// Поддержка соединения
TNC (IN:=NOT Asda.Connect, PT:=T#2S);

CASE CNT OF
0: // Начало работы
	STEP:=0;	// Сброс селектора
	Asda.IsInit:=FALSE;
	Asda.IsHoming:=FALSE;
	Asda.IsServo_ON:=FALSE;
	Asda.Pusk:=FALSE;
	Asda.P2_30:=0;
	Asda.P3_06:=0;
	Asda.E_CODE:=0;
	ALARM_TEST:=FALSE;
	DEL (IN:=FALSE);
	CNT:=10;
	
10: // Ожидание соединения
	Asda.text_id:=12;	// Ожидание соединения
	IF Asda.Connect THEN
		CNT:=20;
	END_IF

20: // Инициализация
	ASDA_INIT (CNT:=STEP);
	IF STEP=0 THEN
		CNT:=TERNAR_INT (Asda.IsInit, 30, 1000);
	END_IF

30: // Запись параметров
	ASDA_PARAMS (CNT:=STEP);
	IF STEP=0 THEN
		CNT:=100;
	END_IF

//////////////////////////////////////////////////////////////////////////////////////////////////
// О Ж И Д А Н И Е  К О М А Н Д Ы  И  Р А З О Г Р Е В А //////////////////////////////////////////
//////////////////////////////////////////////////////////////////////////////////////////////////
100: // Если ручная работа, переход на ручную, иначе Достигла ли температура ? 
	CNT:=PENTAR_INT (Asda.AllowManual, Asda.Block, 180, 110, 130);

110: // Если температура не достигнута, то проверим, включен ли сервопривод, если включен, то отключим
	CNT:=TERNAR_INT (NOT Asda.IsServo_ON, 100, 120);
	
120: // Отключим сервопривод при низких температурах
	ASDA_SERVO_OFF (CNT:=STEP);
	IF STEP=0 THEN
		CNT:=100;
	END_IF
	
130: // Если температура достигнута, то проверим, включен ли сервопривод, если выключен, то включим его
	CNT:=TERNAR_INT (NOT Asda.IsServo_ON, 140, 150);

140: // Включим сервопривод
	ASDA_SERVO_ON (CNT:=STEP);
	IF STEP=0 THEN
		CNT:=150;
	END_IF
	
150: // Проверим Homing, если нет, то выполним Homing
	CNT:=TERNAR_INT (NOT Asda.IsHoming, 160, 170);

160: // Если не было Homing то сделаем Homing
	ASDA_HOMING (CNT:=STEP);
	IF STEP=0 THEN
		CNT:=170;
	END_IF
	
170: // Проверка на запуск
	Asda.text_id:=0; // Индекс сообщения
	CNT:=TERNAR_INT (Asda.Pusk, 200, 100);
	
//////////////////////////////////////////////////////////////////////////////////////////////////
// Р У Ч Н О Й  Р Е Ж И М  ///////////////////////////////////////////////////////////////////////
//////////////////////////////////////////////////////////////////////////////////////////////////
180: // Ручная работа сервопривода - ожидание снятия флага ручной работы
	Asda.text_id:=14;						// Сообщение
	IF NOT Asda.AllowManual THEN
		CNT:=100;
	END_IF
	
//////////////////////////////////////////////////////////////////////////////////////////////////
// О С Н О В Н А Я  Р А Б О Т А //////////////////////////////////////////////////////////////////
//////////////////////////////////////////////////////////////////////////////////////////////////
200: // Пульсирование
	ASDA_PULSING (CNT:=STEP);
	IF STEP=0 THEN
		CNT:=TERNAR_INT (NOT Asda.Block, 210, 100);
	END_IF
	
210: // Парковка
	ASDA_PARKING (CNT:=STEP);
	IF STEP=0 THEN
		CNT:=100;	// На ожидание
	END_IF

//////////////////////////////////////////////////////////////////////////////////////////////////
// О Б Р А Б О Т К А  О Ш И Б О К ////////////////////////////////////////////////////////////////
//////////////////////////////////////////////////////////////////////////////////////////////////
1000: // Сброс
	Asda.DoPulsing:=FALSE;
	STEP:=0;
	DEL (IN:=FALSE);
	CNT:=1010;
	
1010: // Если нет аварии сервопривода, то останов
	CNT:=TERNAR_INT (NOT Asda.E_CODE.0, 1020, 1030);

1020: // Если нет аварии сервопривода, то экстренный стоп
	ASDA_STOP (CNT:=STEP);
	IF STEP=0 THEN
		CNT:=1030;
	END_IF
	
1030: // Ожидание сигнала ОБЩЕГО СБРОСА АВАРИИ или сброса аварии только сервопривода
	Asda.text_id:=10;		// Обработка ошибки
	IF SBROS_AVARII OR SBROS_AVARII_ASDA THEN
		CNT:=TERNAR_INT (Asda.E_CODE.0, 1040, 1050);
	END_IF
	
1040: // Сброс аварии сервопривода
	ASDA_SERVO_ON (CNT:=STEP);
	IF STEP=0 THEN
		CNT:=1050;
	END_IF

1050: // Небольшая задержка
	DEL (IN:=TRUE, PT:=T#1S);
	IF DEL.Q THEN
		DEL (IN:=FALSE);
		CNT:=1060;
	END_IF

1060: // Ожидание пропадания сигнала SBROS_AVARII
	IF NOT (SBROS_AVARII OR SBROS_AVARII_ASDA) THEN
		Asda.IsHoming:=FALSE;
		Asda.E_CODE:=0;
		ALARM_TEST:=FALSE;
		CNT:=100;
	END_IF
	
END_CASE

// Обнаружение пропадания соединения
IF CNT >= 100 AND TNC.Q THEN
	CNT:=0;
	RETURN;
END_IF

// Формирование аппаратных ошибок (программные ошибки формируются внутри обработчиков операций)
IF CNT < 1000 AND NOT Asda.AllowManual THEN
	IF Asda.P0_46.6 THEN Asda.E_CODE.0:=TRUE; END_IF							// ALRM (Авария привода)
	IF Asda.P0_46.10 AND Asda.DoPulsing THEN Asda.E_CODE.1:=TRUE; END_IF		// WARN ()
	IF Asda.P0_46.5 THEN Asda.E_CODE.5:=TRUE; END_IF							// TQL - Сигнал превышения момента
	IF ALARM_TEST THEN Asda.E_CODE.6:=TRUE;	END_IF								// Тестовая ошибка
END_IF

// Блокировка ошибки при ручном режиме
IF Asda.AllowManual THEN
	Asda.E_CODE:=0;
END_IF

// Обнаружение аварий
IF Asda.E_CODE <> 0 AND CNT < 1000 THEN
	CNT:=1000;
END_IF

// Флаг ожидания
Asda.WAIT:=CNT >= 100 AND CNT < 200;
Asda.WAIT_WORK:=CNT >= 200 AND CNT < 1000; 
Asda.WAIT_ERR:=CNT >= 1000;

// Блокируем все сообщения при разогреве
IF CNT >= 100 AND CNT < 1000 AND Asda.Block THEN
	Asda.text_id:=13; // Индекс сообщения "Ожидание температур запуска"
END_IF

END_PROGRAM

// Device/Application/SRC/ASDA_INIT
PROGRAM ASDA_INIT
VAR_IN_OUT
	CNT	: INT;
END_VAR
VAR
	DEL			: TON;
	attempts	: BYTE;

END_VAR


CASE CNT OF
0: // Сначала задержка, чтобы начался обмен данными СПК с устройствами
	Asda.text_id:=1;						// Индекс сообщения
	Asda.IsInit:=FALSE;						// Сброс флага инициализации
	Asda.P2_30:=0;							// Сброс Р2-30
	Asda.P3_06:=0;							// Сброс Р3-06
	attempts:=0;
	DEL (IN:=FALSE);
	CNT:=5;									// Переход

5:	// Проверка Р2-30 и Р3-06
	IF Asda.P2_30=5 AND Asda.P3_06=3 THEN
		Asda.IsInit:=TRUE;					// Установка флага инициализации
		CNT:=90;
	ELSE
		IF attempts = 3 THEN				// Если безушпешные 3 попытки
			Asda.E_CODE.2:=TRUE;				// Ошибка инициализации Р2-30 или Р3-06
			CNT:=100;
		ELSE		
			// Запись Р2-30=5 и Р3-06=3
			AddWriteCmd (wCmd:=wcAsda_P2_30);	// См. фукнцию AddWriteCmd	
			AddWriteCmd (wCmd:=wcAsda_P3_06);	// См. фукнцию AddWriteCmd	
			CNT:=10;							// Переход
		END_IF
	END_IF

10:	// Выдержка времени 1 сек (Чтение P2-30 и P3_06 осуществляется непрерывно с помощью Mapping (см. файл COM1_PRG))
	DEL (IN:=TRUE, PT:=T#1S);
	IF DEL.Q THEN
		DEL (IN:=FALSE);
		CNT:=20;						// Переход
	END_IF

20: // Увеличение счётчика
	attempts:=attempts+1;
	CNT:=5;
	
90:	// Выдержка времени 2 сек
	DEL (IN:=TRUE, PT:=T#2S);
	IF DEL.Q THEN
		DEL (IN:=FALSE);
		CNT:=100;
	END_IF
			
100: // Конец 
	CNT:=0;
	
END_CASE

END_PROGRAM

// Device/Application/SRC/TERNAR_INT
FUNCTION TERNAR_INT : INT
VAR_INPUT
	COND	: BOOL;
	RES1	: INT;
	RES2	: INT;
END_VAR
VAR
END_VAR

IF COND THEN
	TERNAR_INT:=RES1;
ELSE
	TERNAR_INT:=RES2;
END_IF

END_FUNCTION

// Device/Application/SRC/ASDA_PARAMS
PROGRAM ASDA_PARAMS
VAR_IN_OUT
	CNT	: INT;
END_VAR
VAR
	DEL : TON;
	
END_VAR


CASE CNT OF

0:	// Установка индекса сообщения параметров
	Asda.text_id:=9;
	DEL (IN:=FALSE);
	CNT:=10;
	
10:	// Установка параметров сервопривода
	AsdaSetParams ();	// Параметры периода Asda
	CNT:=90;

90:	// Увеличим выдержку времени до 3 сек (ранее было 2 сек)
	DEL (IN:=TRUE, PT:=T#3S);
	IF DEL.Q=0 THEN
		DEL (IN:=FALSE);
		CNT:=100;
	END_IF

100: // Конец 
	CNT:=0;

END_CASE

END_PROGRAM

// Device/Application/SRC/AsdaSetParams
PROGRAM AsdaSetParams
VAR_INPUT
END_VAR
VAR
	dRep		: DINT;
	wSpeeds		: ARRAY [0..1] OF WORD;			// обороты в мин
	wAccs		: ARRAY [0..3] OF WORD;			// обороты в мин
	wDels		: ARRAY [0..1] OF WORD;			// милисекунды
	dOffsets	: ARRAY [0..1] OF DINT;
	dist		: REAL;
	tPeriod		: REAL;			
	tHalfs		: ARRAY [0..1] OF REAL;
	tPulses		: ARRAY [0..1] OF REAL;
	tLevels		: ARRAY [0..1] OF REAL;
	tAccs		: ARRAY [0..1] OF REAL;
	midSpeeds	: ARRAY [0..1] OF REAL;
	vSpeeds		: ARRAY [0..1] OF REAL;
END_VAR


// 1. Сначала записать положение реперной точки P6-01, адрес 16х0602
dRep:=REAL_TO_DINT (Setts.REP_MM * PUU_PER_MM);
QueuePushReg (ADR (COM1_PRG.WR_REGS), ADR_ASDA, 16#0602, ADR (dRep), 2);			// Р6-01 Положение реперной точки

// 2. Запись перемещения 1-го полупериода, т.к. оно используется при вычислении следующих параметров
dOffsets[0]:=REAL_TO_DINT (REG_W.Period.Offsets[0] * PUU_PER_MM);
QueuePushReg (ADR (COM1_PRG.WR_REGS), ADR_ASDA, 16#062A, ADR (dOffsets[0]), 2);	// Р6-21 Смещение 1-го полупериода рабочее
QueuePushReg (ADR (COM1_PRG.WR_REGS), ADR_ASDA, 16#063A, ADR (dOffsets[0]), 2);	// Р6-29 Смещение 1-го полупериода для ШАГА позиционирования 14 (ручное перемещение)

// Запись перемещения 2-го полупериода, т.к. оно используется при вычислении следующих параметров
dOffsets[1]:=REAL_TO_DINT (REG_W.Period.Offsets[1] * PUU_PER_MM);
QueuePushReg (ADR (COM1_PRG.WR_REGS), ADR_ASDA, 16#062E, ADR (dOffsets[1]), 2);	// Р6-23 Смещение 2-го полупериода
QueuePushReg (ADR (COM1_PRG.WR_REGS), ADR_ASDA, 16#063E, ADR (dOffsets[1]), 2);	// Р6-31 Смещение 2-го полупериода для шага позиционирования 15 (ручное перемещение)

// Время периода в секундах
tPeriod:= 1 / REG_W.Freq;
	
// Времена полупериодов в секундах
tHalfs[0]:=tPeriod * REG_W.Period.Per_FirstHP / 100;
tHalfs[1]:=tPeriod - tHalfs[0];
	
// Времена импульсов в секундах
tPulses[0]:=tHalfs[0] * REG_W.Period.Per_Pulses[0] / 100;
tPulses[1]:=tHalfs[1] * REG_W.Period.Per_Pulses[1] / 100;
	
// Фронты полупериодов (импульсов) в секундах - Длина импульса минус длина уровня, делённая на 2
tAccs[0]:=tPulses[0] * (100 - REG_W.Period.Per_Levels[0]) / 200;
tAccs[1]:=tPulses[1] * (100 - REG_W.Period.Per_Levels[1]) / 200;
	
// Уровни полупериодов
tLevels[0]:=tPulses[0] * REG_W.Period.Per_Levels[0] / 100;
tLevels[1]:=tPulses[1] * REG_W.Period.Per_Levels[1] / 100;
	
// Пройденный путь в мм
dist:=ABS (REG_W.Period.Offsets[0] - REG_W.Period.Offsets[1]);
	
// Средние скорости в мм/сек
midSpeeds[0]:=dist / tPulses[0];
midSpeeds[1]:=dist / tPulses[1];
	
// Расчётные скорости в мм/сек
vSpeeds[0]:=midSpeeds[0] * (2 * tAccs[0] + tLevels[0]) / (tAccs[0] + tLevels[0]);
vSpeeds[1]:=midSpeeds[1] * (2 * tAccs[1] + tLevels[1]) / (tAccs[1] + tLevels[1]);
		
// Пересчёт скорости, данные - l оборот => 5 мм перемещения
// 5 мм/сек = 1 об/сек =>
wSpeeds[0]:=REAL_TO_WORD (vSpeeds[0] * 60 * 10 / 5);	// Получили в об/мин (Нужно умножить на 10, т.к. в сервоприводе единица измерения скорости 0.1 об/мин)
wSpeeds[1]:=REAL_TO_WORD (vSpeeds[1] * 60 * 10 / 5);	// Получили в об/мин

// Пересчёт фронт и спада относительно скорости wSpeeds[0]
wAccs[0]:=REAL_TO_WORD (tAccs[0] * 3000 * 1000 / wSpeeds[0]);	
wAccs[1]:=REAL_TO_WORD (tAccs[0] * 3000 * 1000 / wSpeeds[0]);
wAccs[2]:=REAL_TO_WORD (tAccs[1] * 3000 * 1000 / wSpeeds[1]);
wAccs[3]:=REAL_TO_WORD (tAccs[1] * 3000 * 1000 / wSpeeds[1]);
	
// Задержки в миллисекундах
wDels[0]:=REAL_TO_WORD ((tHalfs[0] - tPulses[0]) * 1000.0);
wDels[1]:=REAL_TO_WORD ((tHalfs[1] - tPulses[1]) * 1000.0);

// Запись	
QueuePushReg (ADR (COM1_PRG.WR_REGS), ADR_ASDA, 16#0528, ADR (wAccs[0]), 1);		// Р5-20 Фронт 1-го полупериода
QueuePushReg (ADR (COM1_PRG.WR_REGS), ADR_ASDA, 16#052A, ADR (wAccs[1]), 1);		// Р5-21 Спад 1-го полупериода 
QueuePushReg (ADR (COM1_PRG.WR_REGS), ADR_ASDA, 16#052C, ADR (wAccs[2]), 1);		// Р5-22 Фронт 2-го полупериода
QueuePushReg (ADR (COM1_PRG.WR_REGS), ADR_ASDA, 16#052E, ADR (wAccs[3]), 1);		// Р5-23 Спад 2-го полупериода 

QueuePushReg (ADR (COM1_PRG.WR_REGS), ADR_ASDA, 16#0578, ADR (wSpeeds[0]), 1);		// Р5-60 Скорость 1-го полупериода
QueuePushReg (ADR (COM1_PRG.WR_REGS), ADR_ASDA, 16#057A, ADR (wSpeeds[1]), 1);		// Р5-61 Скорость 2-го полупериода 

QueuePushReg (ADR (COM1_PRG.WR_REGS), ADR_ASDA, 16#0550, ADR (wDels[0]), 1);		// Р5-40 Задержка 1-го полупериода
QueuePushReg (ADR (COM1_PRG.WR_REGS), ADR_ASDA, 16#0552, ADR (wDels[1]), 1);		// Р5-41 Задержка 2-го полупериода

END_PROGRAM

// Device/Application/SRC/PENTAR_INT
FUNCTION PENTAR_INT : INT
VAR_INPUT
	COND1	: BOOL;
	COND2	: BOOL;
	RES1	: INT;
	RES2	: INT;
	RES3	: INT;

END_VAR
VAR
END_VAR

IF COND1 THEN
	PENTAR_INT:=RES1;
ELSIF COND2 THEN
	PENTAR_INT:=RES2;	
ELSE
	PENTAR_INT:=RES3;
END_IF

END_FUNCTION

// Device/Application/SRC/ASDA_SERVO_OFF
PROGRAM ASDA_SERVO_OFF
VAR_IN_OUT
	CNT	: INT;
END_VAR
VAR
	DEL : TON;
	
END_VAR


CASE CNT OF

0: // Начало
	Asda.text_id:=8;				// Индекс сообщения
	DEL (IN:=FALSE);
	CNT:=10;						// Переход

10: // Устанавливаем сигнал СБРОС при выключенном SERVO_ON
	AddWriteCmd (wCmd:=wcAsda_P4_07_3);	// Запись 10 в Р4-07 (сброс ошибок и выключенние servo_off)
	CNT:=20;							// Переход

20:	// Задержка 3 сек
	DEL (IN:=TRUE, PT:=T#3S);
	IF DEL.Q THEN
		DEL (IN:=FALSE);
		CNT:=30;					// Переход
	END_IF

30:	// Сбрасываем сигнал СБРОС при выключенном SERVO_ON
	AddWriteCmd (wCmd:=wcAsda_P4_07_1);	// Запись 00 в Р4-07 (servo_off)
	CNT:=40;							// Переход
	
40:	// Задержка 1 сек
	DEL (IN:=TRUE, PT:=T#1S);
	IF DEL.Q THEN
		DEL (IN:=FALSE);
		CNT:=100;					// Переход
	END_IF

100: // Конец
	Asda.IsServo_ON:=FALSE;
	CNT:=0;
	
END_CASE

END_PROGRAM

// Device/Application/SRC/ASDA_SERVO_ON
PROGRAM ASDA_SERVO_ON
VAR_IN_OUT
	CNT	: INT;
END_VAR
VAR
	DEL : TON;
END_VAR


CASE CNT OF
0: // Начало
	Asda.text_id:=6;	// Индекс сообщения
	DEL (IN:=FALSE);
	CNT:=10;

10: // Устанавливает сигнал СБРОС и SERVO_ON на сервоприводе
	AddWriteCmd (wCmd:=wcAsda_P4_07_4);	// См. функцию AddWriteCmd
	CNT:=20;							// Переход

20:	// Задержка 3 сек
	DEL (IN:=TRUE, PT:=T#3S);
	IF DEL.Q THEN
		DEL (IN:=FALSE);
		CNT:=30;			// Переход
	END_IF

30:	// Сбрасываем сигнал СБРОС при включенном SERVO_ON
	AddWriteCmd (wCmd:=wcAsda_P4_07_2);	// См. функцию AddWriteCmd
	CNT:=40;							// Переход
	
40:	// Задержка 0.5 сек
	DEL (IN:=TRUE, PT:=T#500MS);
	IF DEL.Q THEN
		DEL (IN:=FALSE);
		CNT:=100;					// Переход
	END_IF

100: // Конец
	Asda.IsServo_ON:=TRUE;
	CNT:=0;

END_CASE

END_PROGRAM

// Device/Application/SRC/ASDA_HOMING
PROGRAM ASDA_HOMING
VAR_IN_OUT
	CNT	: INT;
END_VAR
VAR
	DEL : TON;
	DOG : TON;	
	tm_homing	: TIME:=T#10S;
	
END_VAR


CASE CNT OF

0:	// Запуск Homing
	Asda.text_id:=2;						// Сообщение
	Asda.IsHoming:=FALSE;					// Сброс флага нахождения реперной точки
	DOG (IN:=FALSE, PT:=tm_homing);
	DEL (IN:=FALSE);
	IF Asda.IsServo_ON AND NOT Asda.Block THEN
		Asda.text_id:=2;					// Индекс сообщения
		AddWriteCmd (wCmd:=wcAsda_Homing);	// Запуск
		CNT:=10;							// Переход
	ELSE	
		CNT:=100;							// Блокировка выполнения при отсутствии Servo_ON
	END_IF
	
10:	// Ожидание 1 сек пока Р5-07 станет отличным от 20001 (Выполняются 2 программы: PR#0 (homing) и PR#1(позиционирование)
	DEL (IN:=TRUE, PT:=T#2S);
	IF DEL.Q THEN
		DEL (IN:=FALSE);
		CNT:=20;
	END_IF

20: // Ждём пока значение Р5-07 станет равно 20001 - значение окончания HOMING
	IF Asda.P5_07 = 20001 THEN
		CNT:=100;
		Asda.IsHoming:=TRUE;
	END_IF

	// Сторожевой таймер
	DOG (IN:=TRUE, PT:=tm_homing);
	IF DOG.Q THEN
		Asda.E_CODE.3:=TRUE;		// Превышено время операции Homing
		CNT:=100;
	END_IF
	
100: // Завершение
	CNT:=0;

END_CASE

END_PROGRAM

// Device/Application/SRC/ASDA_PULSING
PROGRAM ASDA_PULSING
VAR_IN_OUT
	CNT	: INT;
END_VAR
VAR
	DEL : TON;
	
END_VAR


CASE CNT OF
	
0: 	// Начало
	Asda.text_id:=3;			// Индекс сообщения
	AsdaSetParams ();			// На всякий случай запишем параметры (ПОПРОБУЕМ УБРАТЬ)
	DEL (IN:=FALSE);
	
	CNT:=10;

10:	// Задержка 1 сек
	DEL (IN:=TRUE, PT:=T#1S);
	IF DEL.Q THEN
		DEL (IN:=FALSE);
		CNT:=20;
	END_IF

20:	// Запись команды на пульсирование
	AddWriteCmd (wCmd:=wcAsda_Working);
	CNT:=30;			// Переход
	
25:	// Ждём 500 мс
	DEL (IN:=TRUE, PT:=T#500MS);
	IF DEL.Q THEN
		DEL (IN:=FALSE);
		CNT:=26;
	END_IF
	
26: // Установить флаг DoPulsing
	Asda.DoPulsing:=TRUE;	
	CNT:=30;
	
30: // ЗДЕСЬ ИДЁТ ОСНОВНАЯ РАБОТА

	// Ожидание выключения тумблера "Головка" 
	IF NOT Asda.Pusk THEN
		// Выход при выключении
		CNT:=100;
	END_IF

	IF Asda.Block THEN
		CNT:=100;
	END_IF

100: // Выход (ОСТАНОВ СЕРВОПРИВОДА НЕ ПРОИЗВОДИТСЯ !!!)
	Asda.DoPulsing:=FALSE;
	CNT:=0;

END_CASE

END_PROGRAM

// Device/Application/SRC/ASDA_PARKING
PROGRAM ASDA_PARKING
VAR_IN_OUT
	CNT	: INT;
END_VAR
VAR
	DEL	: TON;
	DOG : TON;
	tm_parking	: TIME:=T#10S;	
	
END_VAR


CASE CNT OF
	
0:	// Сообщение о движении в реперную точку
	DOG (IN:=FALSE, PT:=tm_parking);
	DEL (IN:=FALSE);
	Asda.text_id:=11;						// Сообщение
	IF Asda.IsServo_ON THEN
		AddWriteCmd (wCmd:=wcAsda_Parking);	// Запуск
		CNT:=10;
	ELSE
		CNT:=100;
	END_IF
	
10:	// Ожидание 1 сек пока Р5-07 станет отличным от 20013 (Выполняется программа: PR#13 - парковка
	DEL (IN:=TRUE, PT:=T#1S);
	IF DEL.Q THEN
		DEL (IN:=FALSE);
		CNT:=20;
	END_IF

20: // Ждём пока значение Р5-07 станет равно 20013 - значение окончания HOMING
	IF Asda.P5_07 = 20013 THEN
		CNT:=100;
	END_IF

	// Сторожевой таймер
	DOG (IN:=TRUE, PT:=tm_parking);
	IF DOG.Q THEN
		Asda.E_CODE.4:=TRUE;		// Превышено время операции Parking
		CNT:=100;
	END_IF
	
100: // Завершение
	CNT:=0;

END_CASE

END_PROGRAM

// Device/Application/SRC/ASDA_STOP
PROGRAM ASDA_STOP
VAR_IN_OUT
	CNT	: INT;
END_VAR
VAR
	DEL : TON;
END_VAR


// Экстренный останов
CASE CNT OF
	
0:	// Подаём сигнал экстренного СТОП
	Asda.text_id:=7;	// Индекс сообщения
	AddWriteCmd (wCmd:=wcAsda_Stop); 
	DEL (IN:=FALSE);
	CNT:=10;
	
10:	// Небольшая задержка
	DEL (IN:=TRUE, PT:=T#1S);
	IF DEL.Q THEN
		DEL (IN:=FALSE);
		CNT:=100;
	END_IF

100: // Конец
	CNT:=0;	

END_CASE

END_PROGRAM

// Device/Application/SRC_AUX/SWAP_BYTES
FUNCTION SWAP_BYTES : WORD
VAR_INPUT
	wValue : WORD;
END_VAR
VAR
END_VAR


SWAP_BYTES := SHL (wValue, 8) OR SHR (wValue, 8);

END_FUNCTION

// Device/Application/SRC/AddReadCmd
PROGRAM AddReadCmd
VAR_INPUT
	rCmd	: TReadCmd;
END_VAR

VAR
END_VAR


// В зависимости от команды 
CASE rCmd OF
	//=====================================================================================
	// КОМАНДЫ ДЛЯ ПЕРВОНАЧАЛЬНОЙ ИНИЦИАЛИЗАЦИИ ASDA_A2
	//=====================================================================================
	rcAsda_P2_30	: QueuePushReg (ADR (COM1_PRG.RD_REGS), ADR_ASDA, 16#023C, ADR (Asda.P2_30), 1); 			// Чтение Р2-30 (отключение записи в EEPROM, д.б.= 5)
	rcAsda_P3_06	: QueuePushReg (ADR (COM1_PRG.RD_REGS), ADR_ASDA, 16#030C, ADR (Asda.P3_06), 1); 			// Чтение Р3-06 (способ управления дискретными входами, д.б.= 3)
	
	
END_CASE

END_PROGRAM

// Device/Application/SRC/SET_FRAME_INDEX_EX
FUNCTION SET_FRAME_INDEX_EX : BYTE
VAR_INPUT
	Index : BYTE;
END_VAR
VAR
END_VAR
VAR // added by the converter: edge detectors and wires of the graphical bodies
    _w1 : ANY;
END_VAR

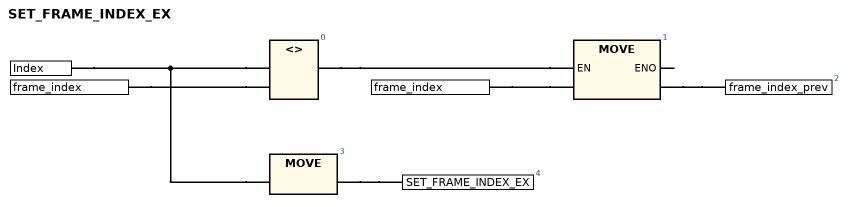
IF Index <> frame_index THEN _w1 := frame_index; END_IF
frame_index_prev := _w1;
SET_FRAME_INDEX_EX := Index;

END_FUNCTION

// Device/Application/SRC/IsRegValid
FUNCTION IsRegValid : BOOL
VAR_INPUT
	pr : POINTER TO TReg;
	
END_VAR
VAR
	I: INT;
END_VAR

IsRegValid:=FALSE;

// Температуры
// Проверка температур
FOR I:=0 TO NUM_TEMPS-1 DO
	IF (pr^.TEMPS[I] < 0) OR (pr^.TEMPS[I] > T_CRITICALS[I]) THEN
		RETURN;
	END_IF
END_FOR

// Температура чиллера
IF (pr^.T_CHIL < 0) OR (pr^.T_CHIL > T_CHIL_CRITICAL) THEN
	RETURN;
END_IF

// Частота колебаний
IF pr^.Freq < FREQ_MIN OR pr^.Freq > FREQ_MAX THEN
	RETURN;
END_IF 

// Смещение 1-го полупериода
IF pr^.Period.Offsets[0] < (Setts.REP_MM + 0.3) OR pr^.Period.Offsets[0] > (WORK_SIZE + Setts.REP_MM - 0.3) THEN
	RETURN;
END_IF

// Смещение 2-го полупериода
IF pr^.Period.Offsets[1] < (Setts.REP_MM + 0.3) OR pr^.Period.Offsets[1] > (WORK_SIZE + Setts.REP_MM - 0.3) THEN
	RETURN;
END_IF

// Проценты полупериодов
IF pr^.Period.Per_FirstHP < ASDA_HP_MIN OR pr^.Period.Per_FirstHP > ASDA_HP_MAX THEN
	RETURN;
END_IF

// Проценты импульсов
IF pr^.Period.Per_Pulses[0] < ASDA_PULSE_MIN OR pr^.Period.Per_Pulses[0] > ASDA_PULSE_MAX THEN
	RETURN;
END_IF

IF pr^.Period.Per_Pulses[1] < ASDA_PULSE_MIN OR pr^.Period.Per_Pulses[1] > ASDA_PULSE_MAX THEN
	RETURN;
END_IF

// Проценты уровня
IF pr^.Period.Per_Levels[0] < ASDA_LEVEL_MIN OR pr^.Period.Per_Levels[0] > ASDA_LEVEL_MAX THEN
	RETURN;
END_IF

IF pr^.Period.Per_Levels[1] < ASDA_LEVEL_MIN OR pr^.Period.Per_Levels[1] > ASDA_LEVEL_MAX THEN
	RETURN;
END_IF

// Скорость заготовки
IF pr^.Speed < SPEED_MIN OR pr^.Speed >= SPEED_MAX THEN
	RETURN;
END_IF

// Производительность
IF pr^.Qm < QM_MIN OR pr^.Qm > QM_MAX THEN
	RETURN;
END_IF

IsRegValid:=TRUE;

END_FUNCTION

// Device/Application/SRC_AUX/BYTES_FROM_DINT
FUNCTION BYTES_FROM_DINT : BOOL
VAR_INPUT
	pBytes	: POINTER TO BYTE;
	iDint	: DINT;
END_VAR
VAR
	pB		: POINTER TO BYTE;
END_VAR

BYTES_FROM_DINT:=TRUE;

pB:=ADR(iDint);

pBytes[0]:=pB[1];
pBytes[1]:=pB[0];
pBytes[2]:=pB[3];
pBytes[3]:=pB[2];

END_FUNCTION

// Device/Application/SRC/MERGE_RGB
FUNCTION MERGE_RGB : DWORD
VAR_INPUT
	clR	: BYTE;
	clG	: BYTE;
	clB	: BYTE;
END_VAR
VAR
END_VAR

MERGE_RGB:=BYTE_TO_DWORD(255);
MERGE_RGB:=SHL(MERGE_RGB,8);
MERGE_RGB:=MERGE_RGB OR BYTE_TO_DWORD(clR);
MERGE_RGB:=SHL(MERGE_RGB,8);
MERGE_RGB:=MERGE_RGB OR BYTE_TO_DWORD(clG);
MERGE_RGB:=SHL(MERGE_RGB,8);
MERGE_RGB:=MERGE_RGB OR BYTE_TO_DWORD(clB);

END_FUNCTION

// Device/Application/SRC_FILE/WRITE_OPTIONS
FUNCTION WRITE_OPTIONS : BOOL
VAR_INPUT
	pSetts	: POINTER TO TSetts;
END_VAR
VAR
	hFile	: SysFile.RTS_IEC_HANDLE;	
	Result	: SysFile.RTS_IEC_RESULT;
	rSize	: __XWORD;
	wrBytes	: __XWORD;
	
END_VAR

WRITE_OPTIONS:=FALSE;

IF NOT MMCMounted THEN
	RETURN;
END_IF

// Создаём новый файл
hFile:=SysFileOpen (OPTIONSFILE, SysFile.AM_WRITE, ADR (Result));
IF Result <> 0 THEN
	RETURN;
END_IF

rSize:=SIZEOF (TSetts);

wrBytes:=SysFileWrite (hFile, pSetts, rSize, ADR (Result));
IF (Result =0 ) AND (wrBytes = rSize) THEN
	WRITE_OPTIONS:=TRUE;
END_IF

SysFileClose (hFile);

END_FUNCTION

// Device/Application/SRC_AUX/HiWord
FUNCTION HiWord : WORD
VAR_INPUT
	dValue	: DINT;
END_VAR	
VAR
	pW		: POINTER TO WORD;
END_VAR

pW:= ADR (dValue);
HiWord:=pW[1];

END_FUNCTION

// Device/Application/SRC_FILE/READ_OPTIONS
FUNCTION READ_OPTIONS : BOOL
VAR_INPUT
	pSetts	: POINTER TO TSetts;
END_VAR
VAR
	hFile	: SysFile.RTS_IEC_HANDLE;	
	Result	: SysFile.RTS_IEC_RESULT;
	fSize	: __XWORD;
	rSize	: __XWORD;
	rdBytes	: __XWORD;
	rdSetts	: TSetts;
	
END_VAR

READ_OPTIONS:=FALSE;

IF NOT MMCMounted THEN
	RETURN;
END_IF


rSize:=SIZEOF (TSetts);

hFile:=SysFileOpen (OPTIONSFILE, SysFile.AM_READ, ADR (Result));
IF Result <> 0 THEN
	RETURN;
END_IF

//  Файл существует, проверяем размер файла
fSize:=SysFileGetSizeByHandle (hFile, ADR (Result));
IF Result <> 0 OR fSize <> rSize THEN
	SysFileClose (hFile);
	RETURN;	
END_IF

rdBytes:=SysFileRead (hFile, ADR (rdSetts), rSize, ADR (Result));	
IF Result = 0 AND rdBytes = rSize THEN
	pSetts^:=rdSetts;
	READ_OPTIONS:=TRUE;
END_IF

SysFileClose (hFile);

END_FUNCTION

// Device/Application/SRC_AUX/LoByte
FUNCTION LoByte : BYTE
VAR_INPUT
	W	: WORD;
END_VAR
VAR
END_VAR

LoByte:=WORD_TO_BYTE (W AND 16#FF);

END_FUNCTION

// Device/Application/SRC_AUX/HiByte
FUNCTION HiByte : BYTE
VAR_INPUT
	W : WORD;
END_VAR
VAR
END_VAR

HiByte:= WORD_TO_BYTE (SHR (W, 8) AND 16#FF);

END_FUNCTION

// Device/Application/SRC_AUX/BYTES_FROM_INT
FUNCTION BYTES_FROM_INT : BOOL
VAR_INPUT
	pBytes	: POINTER TO BYTE;
	vInt	: INT;
END_VAR
VAR
	pB		: POINTER TO BYTE;
END_VAR

BYTES_FROM_INT:=TRUE;

pB:=ADR(vInt);
pBytes[0]:=pB[1];
pBytes[1]:=pB[0];

END_FUNCTION

// Device/Application/SRC/AddWriteCmd_FB
FUNCTION_BLOCK AddWriteCmd_FB
VAR_INPUT
	wcmd	: TWriteCmd;
END_VAR
VAR_OUTPUT
END_VAR
VAR
	
	WR_CMDS			: ARRAY [0..11] OF WORD:=[5, 3, 0, 1, 2, 3, 0, 10, 13, 1000, 14, 15];	// Слова для команд сервопривода
	CH_CMDS			: ARRAY [0..1] OF WORD:=[0, 1];
	// PCHV_CMDS[0],[1] - сформированное управляющее слово для пуска и останова ПЧВ устройств (шнека и тянущего устройства)
	// См. документацию на ПЧВ Овен, а также файл "Управление по RS-485.xlsx",
	// в котором разобраны биты управления и найдены неточности в документации
	SHNEK_CMDS		: ARRAY [0..1] OF WORD:=[1148, 1084];
	PULLING_CMDS	: ARRAY [0..1] OF WORD:=[1148, 1084];
	
	CH_UST			: INT;
	SHNEK_UST		: WORD;
	PULLING_UST		: WORD;

END_VAR

//WR_CMDS[0]:=5;	// Запишем один элемент иначе компилятор не инициализирует правильно массив почему-то, видимо, операция ADR его не устраивает
//CH_CMDS[0]:=0;	// То же

// В зависимости от команды ...
CASE wcmd OF
	//=====================================================================================
	// КОМАНДЫ ПЕРВОНАЧАЛЬНОЙ ИНИЦИАЛИЗАЦИИ
	//=====================================================================================
	wcAsda_P2_30	: QueuePushReg (ADR (COM1_PRG.WR_REGS), ADR_ASDA, 16#023C, ADR (WR_CMDS[0]), 1);	// Параметр  Р2-30 -> 5 (отключение записи в EEPROM) - 5 в старшем байте!
	wcAsda_P3_06	: QueuePushReg (ADR (COM1_PRG.WR_REGS), ADR_ASDA, 16#030C, ADR (WR_CMDS[1]), 1);	// Параметр  Р3-06 -> 3 (способ управления дискретными входами) - 3 в старшем байте!
	wcAsda_P4_07_1	: QueuePushReg (ADR (COM1_PRG.WR_REGS), ADR_ASDA, 16#040E, ADR (WR_CMDS[2]), 1);	// Запись 00 в Р4-07 (servo_off)
	wcAsda_P4_07_2	: QueuePushReg (ADR (COM1_PRG.WR_REGS), ADR_ASDA, 16#040E, ADR (WR_CMDS[3]), 1);	// Запись 01 в Р4-07 (servo_on)
	wcAsda_P4_07_3	: QueuePushReg (ADR (COM1_PRG.WR_REGS), ADR_ASDA, 16#040E, ADR (WR_CMDS[4]), 1);	// Запись 10 в Р4-07 (сброс ошибок и выключенние servo_off)
	wcAsda_P4_07_4	: QueuePushReg (ADR (COM1_PRG.WR_REGS), ADR_ASDA, 16#040E, ADR (WR_CMDS[5]), 1);	// Запись 11 в Р4-07 (сброс ошибок с включенным servo_on)	
	//=====================================================================================
	// КОМАНДЫ УПРАВЛЕНИЯ ASDA
	//=====================================================================================
	wcAsda_Homing	: QueuePushReg (ADR (COM1_PRG.WR_REGS), ADR_ASDA, 16#050E, ADR (WR_CMDS[6]), 1);	// Команда HOMING - запись в Р5-07 числа 0
	wcAsda_Working	: QueuePushReg (ADR (COM1_PRG.WR_REGS), ADR_ASDA, 16#050E, ADR (WR_CMDS[7]), 1);	// Команда WORKING - запись в Р5-07 числа 10
	wcAsda_Parking	: QueuePushReg (ADR (COM1_PRG.WR_REGS), ADR_ASDA, 16#050E, ADR (WR_CMDS[8]), 1);	// Команда PARKING - запись в Р5-07 числа 13
	wcAsda_Stop		: QueuePushReg (ADR (COM1_PRG.WR_REGS), ADR_ASDA, 16#050E, ADR (WR_CMDS[9]), 1);	// КОМАНДА "СТОП" - запись в Р5-07 числа 1000
	wcAsda_Forward	: QueuePushReg (ADR (COM1_PRG.WR_REGS), ADR_ASDA, 16#050E, ADR (WR_CMDS[10]), 1);	// Команда вперёд - запись в Р5-07 числа 14
	wcAsda_Backward	: QueuePushReg (ADR (COM1_PRG.WR_REGS), ADR_ASDA, 16#050E, ADR (WR_CMDS[11]), 1);	// Команда назад - запись в Р5-07 числа 15
	//=====================================================================================
	// КОМАНДА ЗАПИСИ ПАРАМЕТРОВ
	//=====================================================================================

	
	//=====================================================================================
	// КОМАНДЫ ЧИЛЛЕРА
	//=====================================================================================
	wcChiller_Ust:
		CH_UST :=REAL_TO_INT (REG_W.T_CHIL * 10.0);
		QueuePushReg (ADR (COM3_PRG.WR_REGS), ADR_CHILLER, 11, ADR (CH_UST), 1);						// Запись уставки Чиллера

	wcChiller_Start	: QueuePushReg (ADR (COM3_PRG.WR_REGS), ADR_CHILLER, 12, ADR (CH_CMDS[1]), 1);		// Старт Чиллера
	wcChiller_Stop	: QueuePushReg (ADR (COM3_PRG.WR_REGS), ADR_CHILLER, 12, ADR (CH_CMDS[0]), 1);		// Стоп Чиллера

	//=====================================================================================
	// КОМАНДЫ ШНЕКА
	//=====================================================================================
	wcShnek_Ust:
		SHNEK_UST:= REAL_TO_WORD (16382 * REG_W.Qm / 100.0);											// Передаём в частотник число от 0 до 16382 
		QueuePushReg (ADR (COM2_PRG.WR_REGS), ADR_SHNEK, 16#C359, ADR (SHNEK_UST), 1);					// Уставка шнека (ЗАПИСЬ РЕГИСТРА ЗАДАНИЯ REF - РАЗОБРАТЬСЯ !!!)	

	wcShnek_Start: 	QueuePushReg (ADR (COM2_PRG.WR_REGS), ADR_SHNEK, 16#C34F, ADR (SHNEK_CMDS[0]), 1);	// Включение шнека (ЗАПИСЬ УПР.СЛОВА - РАЗОБРАТЬСЯ !!!)
	wcShnek_Stop:	QueuePushReg (ADR (COM2_PRG.WR_REGS), ADR_SHNEK, 16#C34F, ADR (SHNEK_CMDS[1]), 1);	// Выключение шнека (ЗАПИСЬ УПР.СЛОВА - РАЗОБРАТЬСЯ !!!)

	//=====================================================================================
	// КОМАНДЫ ТЯУ
	//=====================================================================================
	wcPulling_Ust:
		PULLING_UST:=REAL_TO_WORD (16382 * REG_W.Speed / 100.0);
		QueuePushReg (ADR (COM2_PRG.WR_REGS), ADR_PULLING, 16#C359, ADR (PULLING_UST), 1);	// Уставка тянущего (ЗАПИСЬ РЕГИСТРА ЗАДАНИЯ REF)

	wcPulling_Start: QueuePushReg (ADR (COM2_PRG.WR_REGS), ADR_PULLING, 16#C34F, ADR (PULLING_CMDS[0]), 1);	// Включение тянущего (ЗАПИСЬ УПР.СЛОВА - РАЗОБРАТЬСЯ !!!)
	wcPulling_Stop:	 QueuePushReg (ADR (COM2_PRG.WR_REGS), ADR_PULLING, 16#C34F, ADR (PULLING_CMDS[1]), 1);	// Выключение тянущего (ЗАПИСЬ УПР.СЛОВА - РАЗОБРАТЬСЯ !!!)


END_CASE

END_FUNCTION_BLOCK

// Device/Application/SRC_FILE/RECORD_SAVE
FUNCTION RECORD_SAVE : BOOL
VAR_INPUT
	pRec	: POINTER TO TReg;
END_VAR
VAR
	hFile	: SysFile.RTS_IEC_HANDLE;	
	Result	: SysFile.RTS_IEC_RESULT;
	fSize	: __XWORD;
	wrBytes	: __XWORD;
	rdBytes	: __XWORD;
	I		: __XWORD;
	rSize	: __XWORD;
	rdRec	: TReg;
	nRec	: __XWORD;
	isOpen	: BOOL;
END_VAR


RECORD_SAVE:=FALSE;
IF NOT MMCMounted THEN
	RETURN;
END_IF

rSize:=SIZEOF (TReg);
isOpen:=FALSE;

// Попытаемся открыть файл saves.dat для чтения и записи
hFile:=SysFileOpen (FILENAME, SysFile.AM_READ_PLUS, ADR( Result));
IF (Result = 0) THEN
	isOpen:=TRUE;
	//  Файл существует, проверяем размер файла
	fSize:=SysFileGetSizeByHandle (hFile, ADR (Result));
	IF (Result = 0) AND (fSize >= rSize) AND ((fSize MOD rSize) = 0) THEN
		nRec:=fSize / rSize;
		//  ищем нужную запись
		FOR I:=0 TO nRec-1 DO
			rdBytes:=SysFileRead(hFile, ADR(rdRec), rSize, ADR(Result));	
			IF (Result=0) AND (rdBytes=rSize) THEN
				IF OSCAT_BASIC.LOWERCASE (pRec^.Name) = OSCAT_BASIC.LOWERCASE (rdRec.Name) THEN
					// Если запись нашли, то переписываем её
					// 1. Позиционируем
					SysFileSetPos (hFile, I * rSize);
					// 2. Записываем из переменной pRec
					wrBytes:=SysFileWrite (hFile, pRec, rSize, ADR (Result));
					IF (Result = 0) AND (wrBytes = rSize) THEN
						SysFileClose (hFile);
 						RECORD_SAVE:=TRUE;
						RETURN;
					END_IF
					
				ELSE	// IF pRec^.Name <> rdRec.Name THEN
					// Если не нашли имя на последней записи, то дописываем в конец
					IF I = (nRec-1) THEN
						wrBytes:=SysFileWrite (hFile, pRec, rSize, ADR (Result));
						IF (Result = 0) AND (wrBytes = rSize) THEN
							SysFileClose (hFile);
	 						RECORD_SAVE:=TRUE;
							RETURN;
						END_IF
					END_IF
				END_IF
			END_IF
		END_FOR
	END_IF
END_IF
 

IF isOpen THEN
	SysFileClose (hFile);
END_IF

// Если не получилось, создаём новый файл
hFile:=SysFileOpen (FILENAME, SysFile.AM_WRITE, ADR(Result));
IF Result = 0 THEN
	wrBytes:=SysFileWrite (hFile, pRec, rSize, ADR (Result));
	IF (Result =0 ) AND (wrBytes = rSize) THEN
		RECORD_SAVE:=TRUE;
	END_IF
	// Закрываем созданный файл
	SysFileClose (hFile);
END_IF

END_FUNCTION

// Device/Application/SRC_FILE/RECS_SELECT
FUNCTION RECS_SELECT : INT												// Число записей на странице (относительное)
VAR_INPUT
	START_INDEX		: INT;												// Стартовый индекс записи (абсолютный)
	OUT_RECS		: POINTER TO ARRAY [0..TABLE_NUM_ROWS-1] OF TREG;	// Выходной массив записей
	NUM_FILE_RECS	: POINTER TO INT;									// Общее число записей в файле
END_VAR
VAR
	hFile	: SysFile.RTS_IEC_HANDLE;	
	Result	: SysFile.RTS_IEC_RESULT;
	fSize	: INT;
	rSize	: INT;
	nRec	: INT;
	nCount	: INT;
	I		: INT;
	
END_VAR

RECS_SELECT:=-1;
NUM_FILE_RECS^:=0;
IF NOT MMCMounted THEN
	RETURN;
END_IF

RECS_SELECT:=-2;
hFile:=SysFileOpen (FILENAME, SysFile.AM_READ, ADR (Result));	// Попытаемся открыть файл saves.dat для чтения
IF Result <> 0 THEN
	RETURN;		//  Если нет, то выходим, считая, что нет рабочего файла
END_IF

RECS_SELECT:=0;

// Размер записи
rSize:=UINT_TO_INT (SIZEOF (TReg));

// Размер файла
fSize:=DWORD_TO_INT (SysFileGetSizeByHandle (hFile, ADR (Result)));
IF (Result <> 0) OR (fSize < rSize) OR ((fsize MOD rSize) <> 0) THEN
	SysFileClose (hFile);
	RETURN;	
END_IF

// Число записей
nRec:=fSize / rSize;  
NUM_FILE_RECS^:=nRec;

IF START_INDEX < nRec THEN
	// Переместим маркер на позицию START_INDEX
	SysFileSetPos (hFile, INT_TO_DWORD (rSize * START_INDEX));
	// Число циклов чтения
	nCount:=MIN (TABLE_NUM_ROWS, nRec - START_INDEX);

	FOR I:=0 TO  nCount-1 DO
		SysFileRead (hFile, ADR (OUT_RECS^[I]), INT_TO_DWORD (rSize), ADR (Result));
		IF (Result <> 0) THEN
			SysFileClose (hFile);
			RETURN;
		END_IF
	END_FOR

	SysFileClose (hFile);
	RECS_SELECT:=nCount;
END_IF

END_FUNCTION

// Device/Application/SRC_FILE/REC_DELETE
FUNCTION REC_DELETE : INT
VAR_INPUT
	pRec	: POINTER TO TREG;
END_VAR
VAR
	hFile	: SysFile.RTS_IEC_HANDLE;	
	Result	: SysFile.RTS_IEC_RESULT;

	thFile	: SysFile.RTS_IEC_HANDLE;	
	tResult	: SysFile.RTS_IEC_RESULT;
	
	rSize	: __XWORD;
	fSize	: __XWORD;
	nRec	: __XWORD;
	I		: __XWORD;
	nCopy	: __XWORD;
	rec		: TREG;
	
END_VAR

REC_DELETE:=0;

IF NOT MMCMounted THEN
	RETURN;
END_IF

hFile:=SysFileOpen (FILENAME, SysFile.AM_READ, ADR(Result));	// Попытаемся открыть файл saves.dat для чтения
IF Result <> 0 THEN
	RETURN;		//  Если нет, то выходим, считая, что нет рабочего файла
END_IF

// Размер записи
rSize:=SIZEOF (TReg);

// Размер файла
fSize:=SysFileGetSizeByHandle (hFile, ADR (Result));
IF (Result <> 0) OR (fSize < rSize) OR ((fsize MOD rSize) <> 0) THEN
	SysFileClose (hFile);
	RETURN;	
END_IF

// Число записей
nRec:=fSize / rSize;  
IF nRec=0 THEN
	SysFileClose (hFile);
	RETURN;	
END_IF

// Создадим временный файл
thFile:=SysFileOpen (TEMPFILE, SysFile.AM_WRITE, ADR (tResult));
IF tResult <> 0 THEN
	SysFileClose (hFile);
	RETURN;	
END_IF

FOR I:=0 TO nRec-1 DO
	// Читаем запись из первого файла
	SysFileRead (hFile, ADR (rec), rSize, ADR (Result));
	IF Result <> 0 THEN
		SysFileClose (hFile);
		SysFileClose (thFile);
		RETURN;
	END_IF
	// Сравниваем с удаляемым, то пропускаем её, т.е. не записываем во временный файл
	IF  OSCAT_BASIC.LOWERCASE (pRec^.Name) = OSCAT_BASIC.LOWERCASE (rec.Name) THEN
		CONTINUE;
	END_IF
	// Если не равна удаляемой, то переписываем запись во временный файл
	SysFileWrite (thFile, ADR (rec), rSize, ADR (tResult));
	IF tResult <> 0 THEN
		SysFileClose (hFile);
		SysFileClose (thFile);
		RETURN;
	END_IF

END_FOR

// Закрываем файлы
SysFileClose (hFile);
SysFileClose (thFile);

Result:=SysFileCopy (FILENAME, TEMPFILE, ADR (nCopy));
IF Result = 0 THEN
	REC_DELETE:=__XWORD_TO_INT (nRec)-1;
END_IF

END_FUNCTION

// Device/Application/SRC_FILE/REC_EXCHANGE
FUNCTION REC_EXCHANGE : BOOL
VAR_INPUT
	INDEX	: INT;
END_VAR
VAR
	hFile	: SysFile.RTS_IEC_HANDLE;	
	Result	: SysFile.RTS_IEC_RESULT;
	fSize	: INT;
	rSize	: INT;
	nRec	: INT;
	Rec		: TReg;
	Rec1	: TReg;
END_VAR

REC_EXCHANGE:=FALSE;
IF NOT MMCMounted THEN
	RETURN;
END_IF

hFile:=SysFileOpen (FILENAME, SysFile.AM_READ, ADR(Result));		// Попытаемся открыть файл saves.dat для чтения
IF Result <> 0 THEN
	RETURN;		//  Если нет, то выходим, считая, что нет рабочего файла
END_IF

// Размер записи
rSize:=UINT_TO_INT (SIZEOF (TReg));

// Размер файла
fSize:= DWORD_TO_INT (SysFileGetSizeByHandle(hFile, ADR (Result)));
IF (Result <> 0) OR (fSize < rSize) OR ((fsize MOD rSize) <> 0) THEN
	SysFileClose (hFile);
	RETURN;	
END_IF

// Число записей
nRec:=fSize / rSize;

// Проверка индекса
IF (INDEX + 1) >= nRec THEN
	SysFileClose (hFile);
	RETURN;	
END_IF

Result:=SysFileSetPos (hFile, INT_TO_DWORD (rSize * INDEX));		// Переместим на позицию INDEX
IF Result <> 0 THEN
	SysFileClose (hFile);
	RETURN;	
END_IF
SysFileRead (hFile, ADR (Rec), INT_TO_DWORD (rSize), ADR (Result));	// Читаем по INDEX в Rec
IF Result <> 0 THEN
	SysFileClose (hFile);
	RETURN;	
END_IF
SysFileRead (hFile, ADR (Rec1), INT_TO_DWORD (rSize), ADR(Result));	// Читаем пр INDEX+1 в Rec1 (следующая запись)
IF Result <> 0 THEN
	SysFileClose (hFile);
	RETURN;	
END_IF
SysFileClose (hFile);									// Закрываем файл

hFile:=SysFileOpen (FILENAME, SysFile.AM_READ_PLUS, ADR (Result));
IF Result <> 0 THEN
	SysFileClose (hFile);
	RETURN;	
END_IF
Result:=SysFileSetPos(hFile, INT_TO_DWORD (rSize * INDEX));			// Переместим на позицию INDEX
IF Result <> 0 THEN
	SysFileClose (hFile);
	RETURN;	
END_IF
SysFileWrite (hFile, ADR (Rec1), INT_TO_DWORD (rSize), ADR (Result));	// Записываем по INDEX в Rec1
IF Result <> 0 THEN
	SysFileClose (hFile);
	RETURN;	
END_IF
SysFileWrite (hFile, ADR (Rec), INT_TO_DWORD (rSize), ADR (Result));	// Записываем по INDEX+1 в Rec
IF Result <> 0 THEN
	SysFileClose (hFile);
	RETURN;	
END_IF
SysFileClose (hFile);												// Закрываем файл

REC_EXCHANGE:=TRUE;

END_FUNCTION

// Device/Application/SRC_FILE/REC_NAME_EXISTS
FUNCTION REC_NAME_EXISTS : BOOL
VAR_INPUT
	recName	: STRING;
END_VAR
VAR
	hFile	: SysFile.RTS_IEC_HANDLE;	
	Result	: SysFile.RTS_IEC_RESULT;

	fSize	: __XWORD;
	rSize	: __XWORD;
	nRec	: __XWORD;
	rdBytes	: __XWORD;
	I		: __XWORD;
	rdRec	: TReg;
	
END_VAR

REC_NAME_EXISTS:=FALSE;
// Проверка наличия ключевого файла
IF NOT MMCMounted THEN
	RETURN;
END_IF

hFile:=SysFileOpen (FILENAME, SysFile.AM_READ, ADR (Result));	// Попытаемся открыть файл
IF Result <> 0 THEN
	RETURN;		//  Если нет, то выходим, считая, что нет рабочего файла
END_IF

// Размер записи
rSize:=SIZEOF (TReg);

// Размер файла
fSize:=SysFileGetSizeByHandle (hFile, ADR (Result));
IF (Result <> 0) OR (fSize < rSize) OR ((fsize MOD rSize) <> 0) THEN
	SysFileClose (hFile);
	RETURN;	
END_IF

// Число записей
nRec:=fSize / rSize;  

// Поиск записи
FOR I:=0 TO nRec-1 DO
	// Читаем очередную запись
	rdBytes:=SysFileRead (hFile, ADR(rdRec), rSize, ADR (Result));
	IF (Result <> 0) OR (rdBytes <> rSize) THEN
		EXIT;
	END_IF
	
	IF OSCAT_BASIC.LOWERCASE (rdRec.Name) = OSCAT_BASIC.LOWERCASE (recName) THEN
		REC_NAME_EXISTS:=TRUE;
		EXIT;
	END_IF
 
END_FOR

SysFileClose (hFile);

END_FUNCTION

// Device/Application/SRC/KEYBOARD_STR
FUNCTION KEYBOARD_STR : BOOL 
VAR_INPUT
	ch			: STRING;					// Добавляемый символ
	pStr		: POINTER TO STRING;		// Указатель на результирующую строку
	pBw			: POINTER TO BOOL;			// 
	shift		: BOOL; 					// Флаг нажатия клавиши Shift
	iStrLen		: INT;	
END_VAR
VAR
	tempStr		: STRING;
END_VAR

IF NOT pBw^ THEN
	pStr^:='';
	pBw^:=TRUE;	
END_IF

IF LEN (pStr^) < iStrLen THEN
	IF shift THEN
		pStr^:=CONCAT (pStr^, OSCAT_BASIC.LOWERCASE (ch));
	ELSE
		pStr^:=CONCAT (pStr^, ch);
	END_IF
END_IF

KEYBOARD_STR:=TRUE;

END_FUNCTION

// Device/Application/SRC/PROCESS_DELAY_FB
FUNCTION_BLOCK PROCESS_DELAY_FB
VAR_INPUT
	del	: TIME;
END_VAR
VAR_IN_OUT
	CNT	: INT;
END_VAR
VAR
	DEL_T 	: TON;
END_VAR


CASE CNT OF
	
0:	// Фронт импульса разжатия прикатки
	DEL_T (IN:=FALSE, PT:=del);
	CNT:=10;
	
10:	// Работает таймер
	DEL_T (IN:=TRUE, PT:=del);
	IF DEL_T.Q THEN
		DEL_T (IN:=FALSE);
		CNT:=20;
	END_IF
	
20:	// Выход
	CNT:=0;
	
END_CASE

END_FUNCTION_BLOCK

// Device/Application/Visu/VIS_SETTS_2
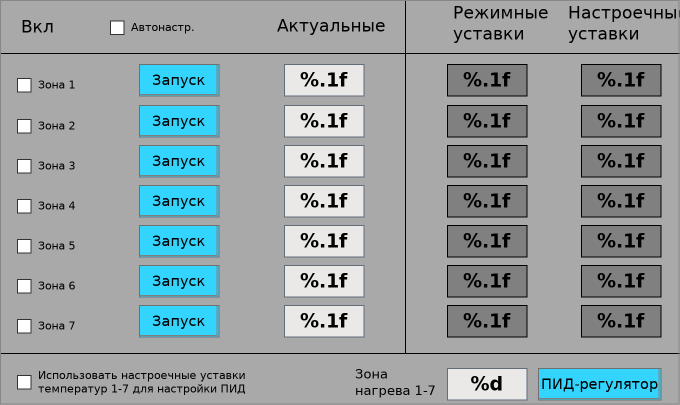
VISUALIZATION VIS_SETTS_2  // 680x405
    Checkbox (15,64 120x42), "Зона 1", variable: Nagrev.T_Enables.0
    Checkbox (15,105 120x42), "Зона 2", variable: Nagrev.T_Enables.1
    Checkbox (15,145 120x42), "Зона 3", variable: Nagrev.T_Enables.2
    Checkbox (15,185 120x42), "Зона 4", variable: Nagrev.T_Enables.3
    Checkbox (15,225 120x42), "Зона 5", variable: Nagrev.T_Enables.4
    Checkbox (15,265 120x42), "Зона 6", variable: Nagrev.T_Enables.5
    Checkbox (15,305 120x42), "Зона 7", variable: Nagrev.T_Enables.6
    Label (18,15 63x24), "Вкл"
    Button (139,64 80x32), "Запуск", colour toggle: Nagrev.Auto_IN.0, input disabled if: NOT Dvp.AutoPIDActivate
        OnMouseClick: execute { Nagrev.Auto_OUT.0:=TRUE; }
    Button (139,105 80x32), "Запуск", colour toggle: Nagrev.Auto_IN.1, input disabled if: NOT Dvp.AutoPIDActivate
        OnMouseClick: execute { Nagrev.Auto_OUT.1:=TRUE; }
    Button (139,145 80x32), "Запуск", colour toggle: Nagrev.Auto_IN.2, input disabled if: NOT Dvp.AutoPIDActivate
        OnMouseClick: execute { Nagrev.Auto_OUT.2:=TRUE; }
    Button (139,185 80x32), "Запуск", colour toggle: Nagrev.Auto_IN.3, input disabled if: NOT Dvp.AutoPIDActivate
        OnMouseClick: execute { Nagrev.Auto_OUT.3:=TRUE; }
    Button (139,225 80x32), "Запуск", colour toggle: Nagrev.Auto_IN.4, input disabled if: NOT Dvp.AutoPIDActivate
        OnMouseClick: execute { Nagrev.Auto_OUT.4:=TRUE; }
    Button (139,265 80x32), "Запуск", colour toggle: Nagrev.Auto_IN.5, input disabled if: NOT Dvp.AutoPIDActivate
        OnMouseClick: execute { Nagrev.Auto_OUT.5:=TRUE; }
    Button (139,305 80x32), "Запуск", colour toggle: Nagrev.Auto_IN.6, input disabled if: NOT Dvp.AutoPIDActivate
        OnMouseClick: execute { Nagrev.Auto_OUT.6:=TRUE; }
    Checkbox (15,361 312x42), "Использовать настроечные уставки температур 1-7 для настройки ПИД", variable: Dvp.zd_selector
    RoundedRectangle (447,64 80x32), "%.1f", text variable: REG_W.TEMPS[0], colour toggle: NOT Dvp.zd_selector
    RoundedRectangle (447,105 80x32), "%.1f", text variable: REG_W.TEMPS[1], colour toggle: NOT Dvp.zd_selector
    RoundedRectangle (447,145 80x32), "%.1f", text variable: REG_W.TEMPS[2], colour toggle: NOT Dvp.zd_selector
    RoundedRectangle (447,185 80x32), "%.1f", text variable: REG_W.TEMPS[3], colour toggle: NOT Dvp.zd_selector
    RoundedRectangle (447,225 80x32), "%.1f", text variable: REG_W.TEMPS[4], colour toggle: NOT Dvp.zd_selector
    RoundedRectangle (447,265 80x32), "%.1f", text variable: REG_W.TEMPS[5], colour toggle: NOT Dvp.zd_selector
    RoundedRectangle (447,305 80x32), "%.1f", text variable: REG_W.TEMPS[6], colour toggle: NOT Dvp.zd_selector
    Label (450,1 107x49), "Режимные уставки"
    RoundedRectangle (581,64 80x32), "%.1f", text variable: Setts.zd_temps[0], colour toggle: Dvp.zd_selector
        OnMouseClick: write the text variable via VisuDialogs.Numpad, min T_MINS_ZAD[6], max T_MAXS_ZAD[6], title "ТЕМПЕРАТУРА 7 ЗОНЫ"
    RoundedRectangle (581,105 80x32), "%.1f", text variable: Setts.zd_temps[1], colour toggle: Dvp.zd_selector
        OnMouseClick: write the text variable via VisuDialogs.Numpad, min T_MINS_ZAD[0], max T_MAXS_ZAD[0]
    RoundedRectangle (581,145 80x32), "%.1f", text variable: Setts.zd_temps[2], colour toggle: Dvp.zd_selector
        OnMouseClick: write the text variable via VisuDialogs.Numpad, min T_MINS_ZAD[0], max T_MAXS_ZAD[0]
    RoundedRectangle (581,185 80x32), "%.1f", text variable: Setts.zd_temps[3], colour toggle: Dvp.zd_selector
        OnMouseClick: write the text variable via VisuDialogs.Numpad, min T_MINS_ZAD[0], max T_MAXS_ZAD[0]
    RoundedRectangle (581,225 80x32), "%.1f", text variable: Setts.zd_temps[4], colour toggle: Dvp.zd_selector
        OnMouseClick: write the text variable via VisuDialogs.Numpad, min T_MINS_ZAD[0], max T_MAXS_ZAD[0]
    RoundedRectangle (581,265 80x32), "%.1f", text variable: Setts.zd_temps[5], colour toggle: Dvp.zd_selector
        OnMouseClick: write the text variable via VisuDialogs.Numpad, min T_MINS_ZAD[0], max T_MAXS_ZAD[0]
    RoundedRectangle (581,305 80x32), "%.1f", text variable: Setts.zd_temps[6], colour toggle: Dvp.zd_selector
        OnMouseClick: write the text variable via VisuDialogs.Numpad, min T_MINS_ZAD[0], max T_MAXS_ZAD[0]
    Label (565,1 127x47), "Настроечные уставки"
    RoundedRectangle (284,64 80x32), "%.1f", text variable: Nagrev.T_Actuals[0], colour variable: Nagrev.FillColors[0]
        p3450524324: Nagrev.FrameColors[0]
    RoundedRectangle (284,105 80x32), "%.1f", text variable: Nagrev.T_Actuals[1], colour variable: Nagrev.FillColors[1]
        p3450524324: Nagrev.FrameColors[1]
    RoundedRectangle (284,145 80x32), "%.1f", text variable: Nagrev.T_Actuals[2], colour variable: Nagrev.FillColors[2]
        p3450524324: Nagrev.FrameColors[2]
    RoundedRectangle (284,185 80x32), "%.1f", text variable: Nagrev.T_Actuals[3], colour variable: Nagrev.FillColors[3]
        p3450524324: Nagrev.FrameColors[3]
    RoundedRectangle (284,225 80x32), "%.1f", text variable: Nagrev.T_Actuals[4], colour variable: Nagrev.FillColors[4]
        p3450524324: Nagrev.FrameColors[4]
    RoundedRectangle (284,265 80x32), "%.1f", text variable: Nagrev.T_Actuals[5], colour variable: Nagrev.FillColors[5]
        p3450524324: Nagrev.FrameColors[5]
    RoundedRectangle (284,305 80x32), "%.1f", text variable: Nagrev.T_Actuals[6], colour variable: Nagrev.FillColors[6]
        p3450524324: Nagrev.FrameColors[6]
    Label (274,14 123x32), "Актуальные"
    Label (352,365 91x40), "Зона нагрева 1-7"
    Button (538,368 123x32), "ПИД-регулятор"
        OnMouseClick:  Dialog=DlgPids, OpenModal=True, OpenCentered=True
    RoundedRectangle (447,368 80x32), "%d", text variable: Dvp.zone_index
        OnMouseClick: write the text variable via VisuDialogs.Numpad, min 1, max 7, title "Введите зону нагрева 1-7"
    Line (405,0) (405,353)
    Line (0,353) (680,353)
    Checkbox (108,9 140x37), "Автонастр.", variable: Dvp.AutoPIDActivate
    Line (0,53) (680,53)
END_VISUALIZATION

// Device/Application/Visu/Main_Panel
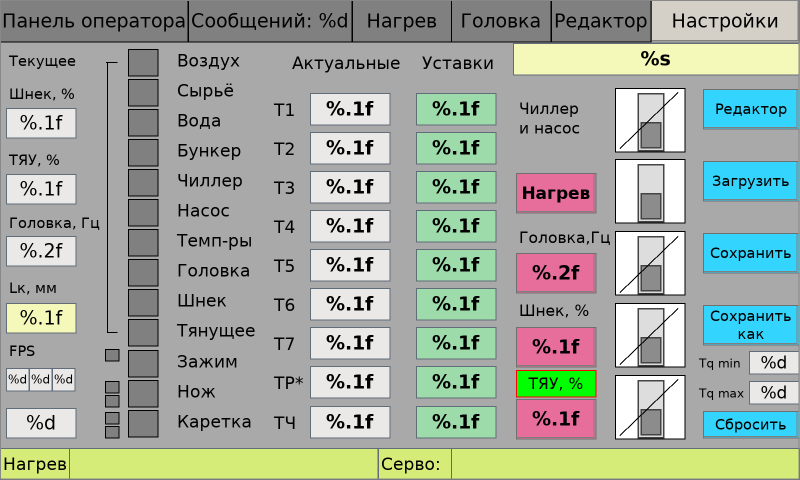
VISUALIZATION Main_Panel  // 800x480
    Rectangle (0,448 80x32), "Нагрев:"
    Frame (94,43 712x442), frame switch variable: frame_index
        shows VIS_OPERATOR()
        shows VIS_MSGS()
        shows VIS_REG()
        shows VIS_PERIOD()
        shows VIS_EDITOR()
    Label (6,213 102x25), "Головка, Гц"
    RoundedRectangle (6,108 70x30), "%.1f", text variable: Shnek.Qm
    Label (6,84 77x27), "Шнек, %"
    Label (6,150 71x26), "ТЯУ, %"
    RoundedRectangle (6,174 70x30), "%.1f", text variable: Pulling.Speed
    Label (6,278 59x25), "Lк, мм"
    RoundedRectangle (6,303 70x30), "%.1f", text variable: Setts.K_Length
        OnMouseClick: write the text variable via VisuDialogs.Numpad, min LEN_MIN, max LEN_MAX, title "Длина заготовки"
    RoundedRectangle (6,236 70x30), "%.2f", text variable: REG_W.Freq
    Label (6,51 79x20), "Текущее"
    Rectangle (0,0 188x42), "Панель оператора", colour toggle: frame_index=0
        OnMouseClick: execute { SET_FRAME_INDEX (0); }
    Rectangle (188,0 164x42), "Сообщений: %d", text variable: alarm_count, colour toggle: frame_index=1
        OnMouseClick: execute { SET_FRAME_INDEX (1); }
    Button (651,0 149x42), "Настройки"
        OnMouseClick:  Assign=Setts_Panel, Type=Assignment
        OnMouseClick: execute {
            parol_vvod:=0; // Сброс ввода пароля
        }
    Rectangle (69,448 309x32), invisible if: CURRENT_PRG.Vigon, text list: 'DvpTextList', text index: Nagrev.text_id
    Rectangle (378,448 80x32), "Серво:"
    Rectangle (451,448 349x32), text list: 'AsdaTextList', text index: Asda.text_id
    RoundedRectangle (6,408 70x30), "%d", text variable: FPS_FULL
    Label (6,341 59x25), "FPS"
    RoundedRectangle (6,368 23x23), "%d", text variable: COM1_PRG.FPS
    RoundedRectangle (29,368 23x23), "%d", text variable: COM2_PRG.FPS
    RoundedRectangle (52,368 23x23), "%d", text variable: COM3_PRG.FPS
    Rectangle (352,0 100x42), "Нагрев", colour toggle: frame_index=2
        OnMouseClick: execute { SET_FRAME_INDEX (2); }
    Rectangle (451,0 100x42), "Головка", colour toggle: frame_index=3
        OnMouseClick: execute { SET_FRAME_INDEX (3); }
    Rectangle (551,0 100x42), "Редактор", colour toggle: frame_index=4
        OnMouseClick: execute { SET_FRAME_INDEX (4); }
END_VISUALIZATION

// Device/Application/Visu/DlgConfirm
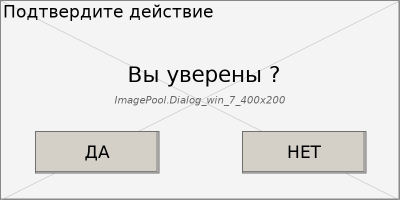
VISUALIZATION DlgConfirm  // 400x200
VAR_IN_OUT
	bDialogVar	: BOOL;
END_VAR
    Image (0,0 400x200), image: ImagePool.Dialog_win_7_400x200
    Button (35,131 124x42), "ДА"
        OnMouseClick:  Dialog=DlgConfirm, Result=OK, NumpadKeypadSet=True
        OnMouseClick: execute { bDialogVar:=TRUE; }
    Button (242,131 124x42), "НЕТ"
        OnMouseClick:  Dialog=DlgConfirm, Result=Cancel, NumpadKeypadSet=True
    Label (80,55 248x39), "Вы уверены ?"
    Label (0,0 248x23), "Подтвердите действие"
END_VISUALIZATION

// Device/Application/Visu/Panel_Reg
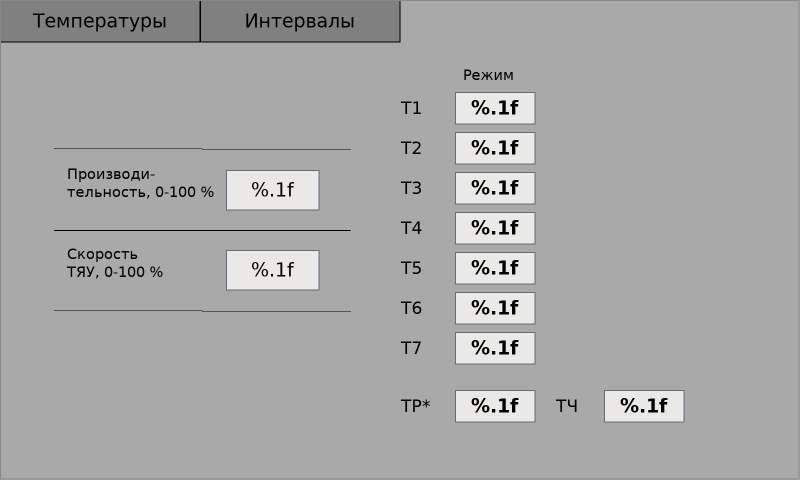
VISUALIZATION Panel_Reg  // 800x480
    Frame (6,47 795x436), frame switch variable: frame_index_reg
        shows VIS_REG()
        shows VIS_PERIOD()
    Rectangle (0,0 200x42), "Температуры", colour toggle: frame_index_reg=0
        OnMouseClick: execute { frame_index_reg:=0; }
    Rectangle (200,0 200x42), "Интервалы", colour toggle: frame_index_reg=1
        OnMouseClick: execute { frame_index_reg:=1; }
END_VISUALIZATION

// Device/Application/Visu/VIS_MSGS
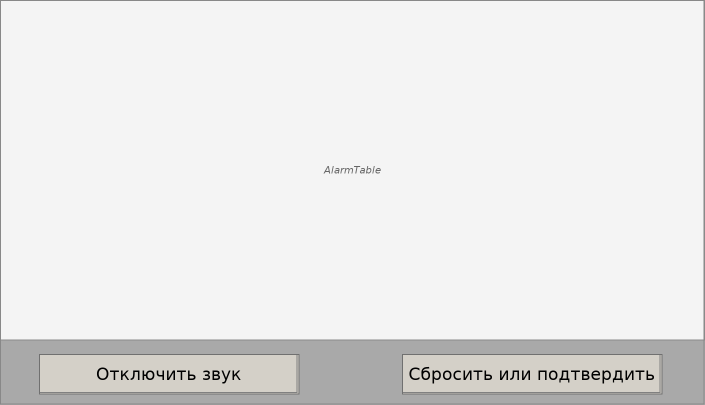
VISUALIZATION VIS_MSGS  // 705x405
VAR_IN_OUT
END_VAR
VAR
	bAckSel : BOOL;
	bAckVisible : BOOL;
	bHistory : BOOL;
	bFreezeScrlPos : BOOL;
END_VAR
    AlarmTable (0,0 705x340)
        Column[0]: ColumnTitle=Изоб
        Column[1]: ColumnTitle=Сообщение
        p1521930926: __All
        p1663851261: __All
        p428520879: bAckSel
        p2607059081: bAckVisible
        p3266827225: bHistory
        p3894972949: bFreezeScrlPos
    Button (39,354 260x40), "Отключить звук", colour toggle: ALARM_ZVUK AND NOT Setts.otkl_alarm_zvuk
        OnMouseClick: execute { ALARM_ZVUK:=FALSE; }
    Button (402,354 260x40), "Сбросить или подтвердить", colour toggle: SBROS_AVARII
        toggle bAckVisible
        OnMouseClick: execute { SBROS_AVARII:=TRUE; }
END_VISUALIZATION

// Device/Application/Visu/VIS_SETTS_4
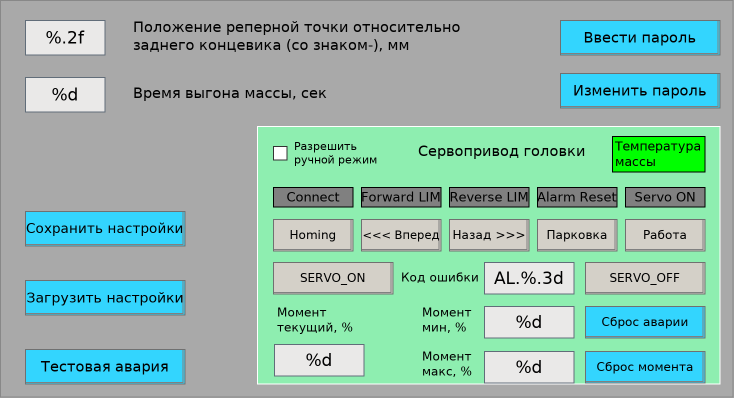
VISUALIZATION VIS_SETTS_4  // 734x398
VAR_IN_OUT

END_VAR

VAR
	bResult : BOOL:=FALSE;
END_VAR
    Rectangle (257,126 463x258)
    Button (25,349 160x35), "Тестовая авария", input disabled if: b_n
        OnMouseClick:  Dialog=DlgConfirm, Parameters={bDialogVar: ALARM_TEST}, Selected={1: }, OpenModal=True, OpenCentered=True
    RoundedRectangle (25,20 80x35), "%.2f", text variable: Setts.REP_MM, input disabled if: b_n
        OnMouseClick: write the text variable via VisuDialogs.Numpad, min REP_MIN, max REP_MAX, title "ЗАДАТЬ РЕПЕРНУЮ ТОЧКУ"
        OnDialogClosed: execute { AsdaSetParams (); }
    Label (130,17 350x52), "Положение реперной точки относительно заднего концевика (со знаком-), мм"
    RoundedRectangle (25,77 80x35), "%d", text variable: Setts.TimeVigon
        OnMouseClick: write the text variable via VisuDialogs.Numpad, min 10, max 10000, title "Время выгона массы в сек"
    Label (130,83 205x28), "Время выгона массы, сек"
    Button (25,211 160x35), "Сохранить настройки", input disabled if: NOT MMCMounted OR b_n
        OnMouseClick:  Dialog=DlgConfirm, Parameters={bDialogVar: bResult}, Selected={1: }, OpenModal=True, OpenCentered=True
        OnDialogClosed: execute {
            IF bResult THEN
            	IF WRITE_OPTIONS (ADR (Setts)) THEN
            		iMsgShowDlg:=5;	// Настройки успешно сохранены
            	ELSE
            		iMsgShowDlg:=6;	// Ошибка при сохранении настроек
            	END_IF
            	CURRENT_PRG.bShowDialog:=TRUE;	// Показать сообщение
            	bResult:=FALSE;
            END_IF
        }
    Button (25,280 160x35), "Загрузить настройки", input disabled if: NOT MMCMounted OR b_n
        OnMouseClick:  Dialog=DlgConfirm, Parameters={bDialogVar: bResult}, Selected={1: }, OpenModal=True, OpenCentered=True
        OnDialogClosed: execute {
            IF bResult THEN
            	IF READ_OPTIONS (ADR (Setts)) THEN
            		iMsgShowDlg:=7;	// Настройки успешно загружены
            	ELSE
            		iMsgShowDlg:=8;	// Ошибка при загрузке настроек
            	END_IF
            	CURRENT_PRG.bShowDialog:=TRUE;	// Показать сообщение
            	bResult:=FALSE;
            END_IF
        }
    Button (560,20 160x35), "Ввести пароль"
        OnMouseClick: write parol_vvod via VisuDialogs.Numpad, min 1, max 65535, title "Введите пароль - число 1-65535"
    Button (560,73 160x35), "Изменить пароль", input disabled if: b_n
        OnMouseClick: write parol via VisuDialogs.Numpad, min 1, max 65535, title "Введите пароль - число 1-65535"
    Label (402,141 200x27), "Сервопривод головки"
    Label (398,269 91x27), "Код ошибки"
    RoundedRectangle (484,262 90x32), "AL.%.3d", text variable: Asda.E_ALARM, colour toggle: Asda.E_ALARM > 0
    Button (585,306 120x32), "Сброс аварии"
        OnMouseClick: execute { SBROS_AVARII_ASDA:=TRUE; }
    Button (273,219 80x32), "Homing", input disabled if: NOT Asda.WAIT OR Asda.Block OR NOT Asda.AllowManual
        OnMouseClick:  Dialog=DlgConfirmAsdaCMD, Parameters={fcmd: wcAsda_Homing}, OpenModal=True, OpenCentered=True
    Button (537,219 80x32), "Парковка", input disabled if: NOT Asda.WAIT OR Asda.Block OR NOT Asda.AllowManual
        OnMouseClick:  Dialog=DlgConfirmAsdaCMD, Parameters={fcmd: wcAsda_Parking}, OpenModal=True, OpenCentered=True
    Button (625,219 80x32), "Работа", input disabled if: NOT Asda.WAIT OR Asda.Block OR NOT Asda.AllowManual
        OnMouseClick:  Dialog=DlgConfirmAsdaCMD, Parameters={fcmd: wcAsda_Working}, OpenModal=True, OpenCentered=True
    Button (361,219 80x32), "<<< Вперед", input disabled if: NOT Asda.WAIT OR Asda.Block OR NOT Asda.AllowManual
        OnMouseClick:  Dialog=DlgConfirmAsdaCMD, Parameters={fcmd: wcAsda_Forward}, OpenModal=True, OpenCentered=True
    Button (449,219 80x32), "Назад >>>", input disabled if: NOT Asda.WAIT OR Asda.Block OR NOT Asda.AllowManual
        OnMouseClick:  Dialog=DlgConfirmAsdaCMD, Parameters={fcmd: wcAsda_Backward}, OpenModal=True, OpenCentered=True
    RoundedRectangle (273,187 80x20), "Connect", colour toggle: Asda.Connect
    RoundedRectangle (537,187 80x20), "Alarm Reset", colour toggle: Asda.P4_07.1
    RoundedRectangle (625,187 80x20), "Servo ON", colour toggle: Asda.P4_07.0
    RoundedRectangle (449,187 80x20), "Reverse LIM", colour toggle: Asda.P4_07.2
    RoundedRectangle (361,187 80x20), "Forward LIM", colour toggle: Asda.P4_07.3
    Label (274,304 91x40), "Момент текущий, %"
    RoundedRectangle (274,344 90x32), "%d", text variable: Asda.Torque
    Button (585,262 120x32), "SERVO_OFF", input disabled if: b_n
        OnMouseClick:  Dialog=DlgConfirmAsdaCMD, Parameters={fcmd: wcAsda_P4_07_1}, OpenModal=True, OpenCentered=True
    Button (273,262 120x32), "SERVO_ON", input disabled if: b_n
        OnMouseClick:  Dialog=DlgConfirmAsdaCMD, Parameters={fcmd: wcAsda_P4_07_2}, OpenModal=True, OpenCentered=True
    Checkbox (271,132 148x42), "Разрешить ручной режим", variable: Asda.AllowManual, input disabled if: NOT Asda.WAIT OR b_n
    RoundedRectangle (612,136 93x36), "Температура массы", colour toggle: Asda.Block
    RoundedRectangle (484,306 90x32), "%d", text variable: Asda.TorqueMin
    Label (419,304 65x36), "Момент мин, %"
    Button (585,351 120x32), "Сброс момента"
        OnMouseClick: execute { Asda.TorqueMin:=0; Asda.TorqueMax:=0; }
    Label (419,348 65x36), "Момент макс, %"
    RoundedRectangle (484,351 90x32), "%d", text variable: Asda.TorqueMax
END_VISUALIZATION

// Device/Application/Visu/Setts_Panel
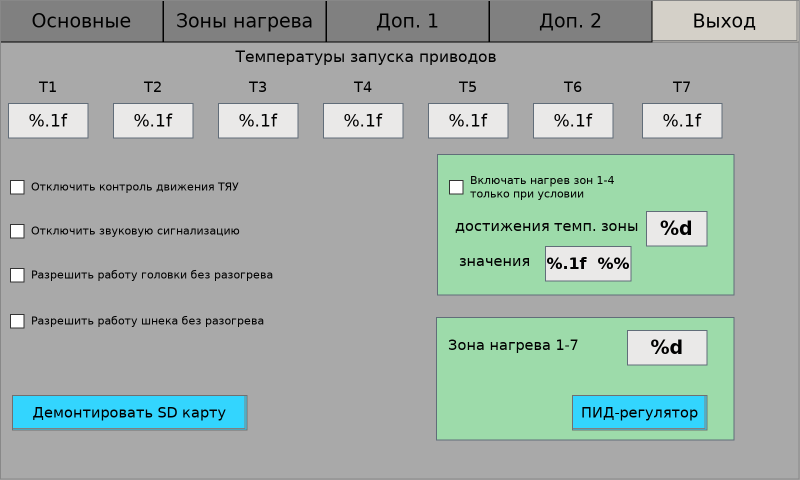
VISUALIZATION Setts_Panel  // 800x480
    Button (650,0 149x42), "Выход"
        OnMouseClick:  Assign=Main_Panel, Type=Assignment
    Rectangle (0,0 163x42), "Основные", colour toggle: frame_index_setts=0
        OnMouseClick: execute { frame_index_setts:=0; }
    Rectangle (163,0 163x42), "Зоны нагрева", colour toggle: frame_index_setts=1
        OnMouseClick: execute { frame_index_setts:=1; }
    Frame (0,43 797x430), frame switch variable: frame_index_setts
        shows VIS_SETTS_1()
        shows VIS_SETTS_2()
        shows VIS_SETTS_3()
        shows VIS_SETTS_4()
    Rectangle (326,0 163x42), "Доп. 1", colour toggle: frame_index_setts=2
        OnMouseClick: execute { frame_index_setts:=2; }
    Rectangle (489,0 163x42), "Доп. 2", colour toggle: frame_index_setts=3
        OnMouseClick: execute { frame_index_setts:=3; }
END_VISUALIZATION

// Device/Application/Visu/VIS_REG
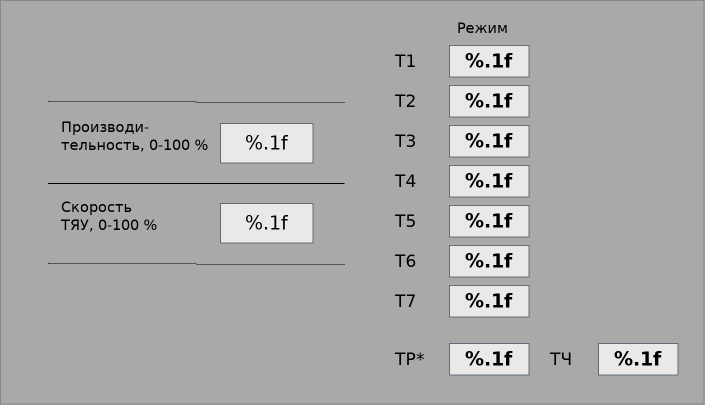
VISUALIZATION VIS_REG  // 705x405
    Line (48,263) (344,264)
    Line (48,183) (344,183)
    Line (48,101) (344,102)
    Label (58,117 162x53), "Производи- тельность, 0-100 %"
    Label (58,197 167x50), "Скорость ТЯУ, 0-100 %"
    RoundedRectangle (220,203 93x40), "%.1f", text variable: REG_W.Speed
        OnMouseClick: write the text variable via VisuDialogs.Numpad, min SPEED_MIN, max SPEED_MAX, title "Скорость заготовки, мм/сек"
    RoundedRectangle (449,45 80x32), "%.1f", text variable: REG_W.TEMPS[0]
        OnMouseClick: write the text variable via VisuDialogs.Numpad, min T_MINS_ZAD[0], max T_MAXS_ZAD[0], title "ТЕМПЕРАТУРА 1 ЗОНЫ"
    Label (392,45 40x32), "T1"
    RoundedRectangle (449,85 80x32), "%.1f", text variable: REG_W.TEMPS[1]
        OnMouseClick: write the text variable via VisuDialogs.Numpad, min T_MINS_ZAD[1], max T_MAXS_ZAD[1], title "ТЕМПЕРАТУРА 2 ЗОНЫ"
    Label (392,85 40x32), "T2"
    RoundedRectangle (449,125 80x32), "%.1f", text variable: REG_W.TEMPS[2]
        OnMouseClick: write the text variable via VisuDialogs.Numpad, min T_MINS_ZAD[2], max T_MAXS_ZAD[2], title "ТЕМПЕРАТУРА3 ЗОНЫ"
    Label (392,125 40x32), "T3"
    RoundedRectangle (449,165 80x32), "%.1f", text variable: REG_W.TEMPS[3]
        OnMouseClick: write the text variable via VisuDialogs.Numpad, min T_MINS_ZAD[3], max T_MAXS_ZAD[3], title "ТЕМПЕРАТУРА 4 ЗОНЫ"
    Label (392,165 40x32), "T4"
    RoundedRectangle (449,205 80x32), "%.1f", text variable: REG_W.TEMPS[4]
        OnMouseClick: write the text variable via VisuDialogs.Numpad, min T_MINS_ZAD[4], max T_MAXS_ZAD[4], title "ТЕМПЕРАТУРА 5 ЗОНЫ"
    Label (392,205 40x32), "T5"
    RoundedRectangle (449,245 80x32), "%.1f", text variable: REG_W.TEMPS[5]
        OnMouseClick: write the text variable via VisuDialogs.Numpad, min T_MINS_ZAD[5], max T_MAXS_ZAD[5], title "ТЕМПЕРАТУРА 6 ЗОНЫ"
    Label (392,245 40x32), "T6"
    RoundedRectangle (449,285 80x32), "%.1f", text variable: REG_W.TEMPS[6]
        OnMouseClick: write the text variable via VisuDialogs.Numpad, min T_MINS_ZAD[6], max T_MAXS_ZAD[6], title "ТЕМПЕРАТУРА 7 ЗОНЫ"
    Label (392,285 40x32), "T7"
    RoundedRectangle (449,343 80x32), "%.1f", text variable: REG_W.T_MASS
        OnMouseClick: write the text variable via VisuDialogs.Numpad, min T_MIN_MASS_ZAD, max T_MAX_MASS_ZAD, title "ТЕМПЕРАТУРА РАСПЛАВА"
    Label (392,343 40x32), "TР*"
    RoundedRectangle (598,343 80x32), "%.1f", text variable: REG_W.T_CHIL
        OnMouseClick: write the text variable via VisuDialogs.Numpad, min T_MIN_CHIL_ZAD, max T_MAX_CHIL_ZAD, title "ТЕМПЕРАТУРА ЧИЛЛЕРА"
    Label (541,343 40x32), "TЧ"
    Label (454,13 76x30), "Режим"
    RoundedRectangle (220,123 93x40), "%.1f", text variable: REG_W.Qm
        OnMouseClick: write the text variable via VisuDialogs.Numpad, min QM_MIN, max QM_MAX, title "Производительность, %"
END_VISUALIZATION

// Device/Application/Visu/VIS_PERIOD
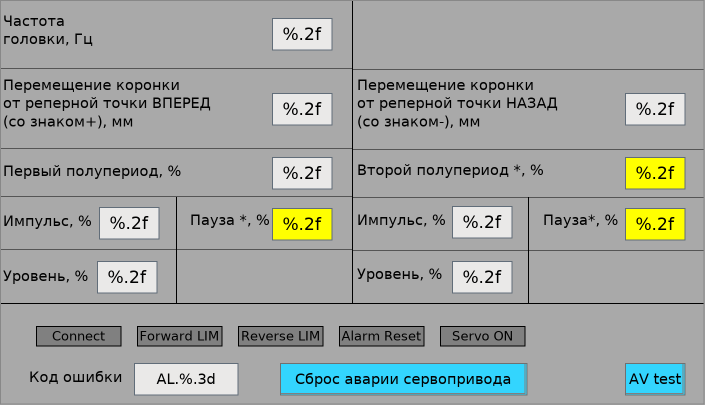
VISUALIZATION VIS_PERIOD  // 705x405
    Label (0,266 102x25), "Уровень, %"
    RoundedRectangle (97,261 60x32), "%.2f", text variable: REG_W.Period.Per_Levels[0]
        OnMouseClick: write the text variable via VisuDialogs.Numpad, min ASDA_LEVEL_MIN, max ASDA_LEVEL_MAX, title "УРОВЕНЬ ПЕРВОГО П/П"
        OnDialogClosed: execute { AsdaSetParams (); }
    RoundedRectangle (452,261 60x32), "%.2f", text variable: REG_W.Period.Per_Levels[1]
        OnMouseClick: write the text variable via VisuDialogs.Numpad, min ASDA_LEVEL_MIN, max ASDA_LEVEL_MAX, title "УРОВЕНЬ ВТОРОГО П/П"
        OnDialogClosed: execute { AsdaSetParams (); }
    Label (0,75 251x72), "Перемещение коронки от реперной точки ВПЕРЕД (со знаком+), мм"
    RoundedRectangle (272,93 60x32), "%.2f", text variable: REG_W.Period.Offsets[0]
        OnMouseClick: write the text variable via VisuDialogs.Numpad, min Setts.REP_MM + 0.3, max WORK_SIZE + Setts.REP_MM - 0.3, title "ПЕРЕМЕЩЕНИЕ 1-ГО П/П"
        OnDialogClosed: execute { AsdaSetParams (); }
    Label (354,75 233x71), "Перемещение коронки от реперной точки НАЗАД (со знаком-), мм"
    RoundedRectangle (625,93 60x32), "%.2f", text variable: REG_W.Period.Offsets[1]
        OnMouseClick: write the text variable via VisuDialogs.Numpad, min Setts.REP_MM + 0.3, max WORK_SIZE + Setts.REP_MM - 0.3, title "ПЕРЕМЕЩЕНИЕ 2-ГО П/П"
        OnDialogClosed: execute { AsdaSetParams (); }
    Line (0,68) (704,69)
    Line (0,303) (704,303)
    Line (0,196) (704,197)
    Label (0,161 214x23), "Первый полупериод, %"
    Label (354,160 216x23), "Второй полупериод *, %"
    Label (354,264 97x25), "Уровень, %"
    Line (352,0) (352,303)
    RoundedRectangle (272,157 60x32), "%.2f", text variable: REG_W.Period.Per_FirstHP
        OnMouseClick: write the text variable via VisuDialogs.Numpad, min ASDA_HP_MIN, max ASDA_HP_MAX, title "ПЕРВЫЙ ПОЛУПЕРИОД"
        OnDialogClosed: execute { AsdaSetParams (); }
    RoundedRectangle (625,157 60x32), "%.2f", text variable: 100 - REG_W.Period.Per_FirstHP
    Line (0,249) (704,250)
    Line (176,197) (176,303)
    RoundedRectangle (99,207 60x32), "%.2f", text variable: REG_W.Period.Per_Pulses[0]
        OnMouseClick: write the text variable via VisuDialogs.Numpad, min ASDA_PULSE_MIN, max ASDA_PULSE_MAX, title "ИМПУЛЬС 1 ПОЛУПЕРИОДА"
        OnDialogClosed: execute { AsdaSetParams (); }
    Label (0,211 94x23), "Импульс, %"
    Label (187,210 94x23), "Пауза *, %"
    RoundedRectangle (272,208 60x32), "%.2f", text variable: 100-REG_W.Period.Per_Pulses[0]
    Label (354,210 94x23), "Импульс, %"
    RoundedRectangle (452,206 60x32), "%.2f", text variable: REG_W.Period.Per_Pulses[1]
        OnMouseClick: write the text variable via VisuDialogs.Numpad, min ASDA_PULSE_MIN, max ASDA_PULSE_MAX, title "ИМПУЛЬС 2 ПОЛУПЕРИОДА"
        OnDialogClosed: execute { AsdaSetParams (); }
    Label (540,210 94x23), "Пауза*, %"
    RoundedRectangle (625,208 60x32), "%.2f", text variable: 100-REG_W.Period.Per_Pulses[1]
    Line (528,197) (528,303)
    Line (0,148) (704,149)
    RoundedRectangle (36,326 85x20), "Connect", colour toggle: Asda.Connect
    RoundedRectangle (339,326 85x20), "Alarm Reset", colour toggle: Asda.P4_07.1
    RoundedRectangle (440,326 85x20), "Servo ON", colour toggle: Asda.P4_07.0
    RoundedRectangle (238,326 85x20), "Reverse LIM", colour toggle: Asda.P4_07.2
    RoundedRectangle (137,326 85x20), "Forward LIM", colour toggle: Asda.P4_07.3
    Label (0,11 144x42), "Частота головки, Гц"
    RoundedRectangle (272,18 60x32), "%.2f", text variable: REG_W.Freq
        OnMouseClick: write the text variable via VisuDialogs.Numpad, min FREQ_MIN, max FREQ_MAX, title "ЧАСТОТА ГОЛОВКИ, Гц"
        OnDialogClosed: execute { AsdaSetParams (); }
    Label (26,367 105x27), "Код ошибки"
    RoundedRectangle (134,363 104x32), "AL.%.3d", text variable: Asda.E_ALARM, colour toggle: Asda.E_ALARM > 0
    Button (280,363 247x32), "Сброс аварии сервопривода"
        OnMouseClick: execute { SBROS_AVARII_ASDA:=TRUE; }
    Button (625,363 60x32), "AV test"
        OnMouseClick:  Dialog=DlgConfirm, Parameters={bDialogVar: ALARM_TEST}, Selected={1: }, OpenModal=True, OpenCentered=True
END_VISUALIZATION

// Device/Application/Visu/VIS_OPERATOR
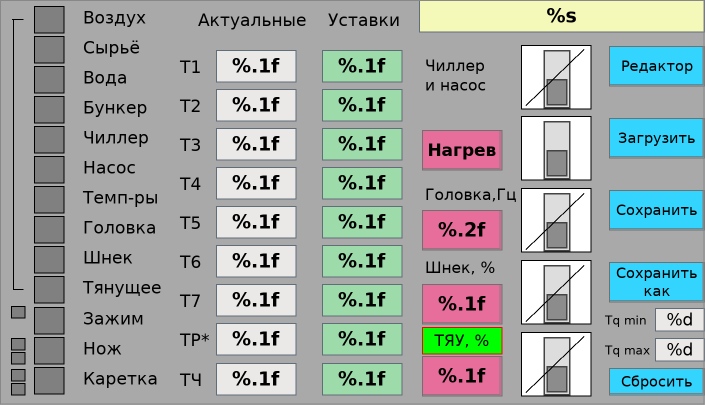
VISUALIZATION VIS_OPERATOR  // 705x405
VAR_IN_OUT

END_VAR

VAR
	iCount: INT;
END_VAR
    RoundedRectangle (521,116 70x64), colour variable: Nagrev.NagrevFillColor
        p3450524324: Nagrev.NagrevFrameColor
    DipSwitch (528,121 58x58), variable: Nagrev.Nagrev_on, behaviour: TOGGLE, style: Switch-DipSwitch-Gray
    RoundedRectangle (521,332 70x64), colour variable: Pulling.BtnFillColor
        p3450524324: Pulling.BtnFrameColor
    DipSwitch (528,337 58x58), variable: Pulling.Pusk, input disabled if: Pulling.Block, behaviour: TOGGLE, style: Switch-DipSwitch-Gray
    RoundedRectangle (521,260 70x64), colour variable: Shnek.FillColor
        p3450524324: Shnek.FrameColor
    DipSwitch (528,265 58x58), variable: Shnek.Pusk, input disabled if: Shnek.Block, behaviour: TOGGLE, style: Switch-DipSwitch-Gray
    RoundedRectangle (521,188 70x64), colour variable: Asda.BtnFillColor
        p3450524324: Asda.BtnFrameColor
    DipSwitch (528,193 58x58), variable: Asda.Pusk, input disabled if: Asda.Block, behaviour: TOGGLE, style: Switch-DipSwitch-Gray
    RoundedRectangle (216,50 80x32), "%.1f", text variable: Nagrev.T_Actuals[0], colour variable: Nagrev.FillColors[0]
        p3450524324: Nagrev.FrameColors[0]
    Label (177,51 40x32), "T1"
    RoundedRectangle (322,50 80x32), "%.1f", text variable: TEMPERS[0], colour toggle: Nagrev.Auto_IN.0
    RoundedRectangle (322,89 80x32), "%.1f", text variable: TEMPERS[1], colour toggle: Nagrev.Auto_IN.1
    RoundedRectangle (216,89 80x32), "%.1f", text variable: Nagrev.T_Actuals[1], colour variable: Nagrev.FillColors[1]
        p3450524324: Nagrev.FrameColors[1]
    Label (177,90 40x32), "T2"
    RoundedRectangle (322,128 80x32), "%.1f", text variable: TEMPERS[2], colour toggle: Nagrev.Auto_IN.2
    RoundedRectangle (216,128 80x32), "%.1f", text variable: Nagrev.T_Actuals[2], colour variable: Nagrev.FillColors[2]
        p3450524324: Nagrev.FrameColors[2]
    Label (177,129 40x32), "T3"
    RoundedRectangle (322,167 80x32), "%.1f", text variable: TEMPERS[3], colour toggle: Nagrev.Auto_IN.3
    RoundedRectangle (216,167 80x32), "%.1f", text variable: Nagrev.T_Actuals[3], colour variable: Nagrev.FillColors[3]
        p3450524324: Nagrev.FrameColors[3]
    Label (177,168 40x32), "T4"
    RoundedRectangle (322,206 80x32), "%.1f", text variable: TEMPERS[4], colour toggle: Nagrev.Auto_IN.4
    RoundedRectangle (216,206 80x32), "%.1f", text variable: Nagrev.T_Actuals[4], colour variable: Nagrev.FillColors[4]
        p3450524324: Nagrev.FrameColors[4]
    Label (177,207 40x32), "T5"
    RoundedRectangle (322,245 80x32), "%.1f", text variable: TEMPERS[5], colour toggle: Nagrev.Auto_IN.5
    RoundedRectangle (216,245 80x32), "%.1f", text variable: Nagrev.T_Actuals[5], colour variable: Nagrev.FillColors[5]
        p3450524324: Nagrev.FrameColors[5]
    Label (177,246 40x32), "T6"
    RoundedRectangle (322,284 80x32), "%.1f", text variable: TEMPERS[6], colour toggle: Nagrev.Auto_IN.6
    RoundedRectangle (216,284 80x32), "%.1f", text variable: Nagrev.T_Actuals[6], colour variable: Nagrev.FillColors[6]
        p3450524324: Nagrev.FrameColors[6]
    Label (177,285 40x32), "T7"
    RoundedRectangle (322,323 80x32), "%.1f", text variable: REG_W.T_MASS
    RoundedRectangle (216,323 80x32), "%.1f", text variable: Nagrev.T_ActualMass, colour variable: Nagrev.FillColorMass
        p3450524324: Nagrev.FrameColorMass
    Label (177,324 48x32), "TР*"
    RoundedRectangle (322,363 80x32), "%.1f", text variable: REG_W.T_CHIL
    RoundedRectangle (216,363 80x32), "%.1f", text variable: Chiller.T_ACTUAL, colour variable: Chiller.FillColor
        p3450524324: Chiller.FrameColor
    Label (177,364 40x32), "TЧ"
    RoundedRectangle (34,186 30x27), colour toggle: Nagrev.Temper_Reached
    Label (80,186 89x32), "Tемп-ры"
    RoundedRectangle (34,216 30x27), colour toggle: Asda.Pusk
    Label (80,216 89x32), "Головка"
    RoundedRectangle (34,246 30x27), colour toggle: Shnek.Pusk
    Label (80,246 89x32), "Шнек"
    RoundedRectangle (34,276 30x27), colour toggle: Pulling.Pusk
    Label (80,276 89x32), "Тянущее"
    RoundedRectangle (34,6 30x27), colour toggle: Dvp.PVozd_si
    Label (80,6 89x32), "Воздух"
    RoundedRectangle (34,156 30x27), colour toggle: Dvp.Nasos_si
    Label (80,156 89x32), "Насос"
    RoundedRectangle (34,36 30x27), colour toggle: Dvp.Uroven_s_si
    Label (80,36 89x32), "Сырьё"
    RoundedRectangle (34,96 30x27), colour toggle: Dvp.Bunker_si
    Label (80,96 89x32), "Бункер"
    RoundedRectangle (521,45 70x64), colour variable: Chiller.BtnFillColor
        p3450524324: Chiller.BtnFrameColor
    DipSwitch (528,50 58x58), variable: Chiller.Pusk, input disabled if: Chiller.Block, behaviour: TOGGLE, style: Switch-DipSwitch-Gray
    Label (422,54 103x43), "Чиллер и насос"
    Line (526,321) (584,265), invisible if: NOT Shnek.Block
    Line (526,392) (584,336), invisible if: NOT Pulling.Block
    Line (526,249) (584,193), invisible if: NOT Asda.Block
    Line (526,105) (584,49), invisible if: NOT Chiller.Block
    RoundedRectangle (34,126 30x27), colour toggle: Chiller.Connect AND Chiller.Status.0
    Label (80,126 89x32), "Чиллер"
    Button (422,130 80x40), "Нагрев"
        OnMouseClick: execute { SET_FRAME_INDEX (2); }
    Button (422,210 80x40), "%.2f", text variable: REG_W.Freq
        OnDialogClosed: execute { AsdaSetParams (); }
        OnMouseClick: write the text variable via VisuDialogs.Numpad, min FREQ_MIN, max FREQ_MAX, title "Частота головки, Гц"
    Label (422,257 91x33), "Шнек, %"
    Label (80,307 89x32), "Зажим"
    RoundedRectangle (34,307 30x27), colour toggle: Dvp.Zazh_si
    Label (80,337 46x32), "Нож"
    RoundedRectangle (34,337 30x27), colour toggle: Dvp.Knife_si
    Label (80,367 89x32), "Каретка"
    RoundedRectangle (34,367 30x27), colour toggle: Dvp.Karet_si
    RoundedRectangle (11,306 14x12), colour toggle: Dvp.ZazhIsx_si
    RoundedRectangle (11,338 14x12), colour toggle: Dvp.KnifeIsx_si
    RoundedRectangle (11,352 14x12), colour toggle: Dvp.KnifeRab_si
    RoundedRectangle (11,369 14x12), colour toggle: Dvp.KarIsx_si
    RoundedRectangle (11,383 14x12), colour toggle: Dvp.KarRab_si
    Label (325,4 80x32), "Уставки"
    Label (191,4 123x32), "Актуальные"
    Line (13,19) (13,289)
    Line (12,19) (23,19)
    Line (13,289) (23,289)
    Button (422,356 80x40), "%.1f", text variable: REG_W.Speed
        OnMouseClick: write the text variable via VisuDialogs.Numpad, min SPEED_MIN, max SPEED_MAX, title "Скорость ТЯУ, %"
    RoundedRectangle (34,66 30x27), colour toggle: Dvp.Uroven_w_si
    Label (80,66 89x32), "Вода"
    Button (422,284 80x40), "%.1f", text variable: REG_W.Qm
        OnMouseClick:  Dialog=DlgTargetRegParams, Parameters={Adapted: , fQm_old: , fFreq: REG_W.Freq, bQm: , fSpeed: REG_W.Speed, fQm: REG_W.Qm}, Selected={1: }, OpenModal=True, OpenCentered=True
    Button (609,118 96x40), "Загрузить", text variable: REG_W.Name, input disabled if: NOT MMCMounted
        OnMouseDown: execute {
            iCount:=RECS_SELECT (0, ADR (TBL.Recs), ADR (TBL.NumFileRecs));
            IF iCount > 0 THEN
            	TBL.RowCount:=iCount;
            	TBL.RowSel:=-32768;			// Сброс выбора строки
            	TBL.PageNum:=0;				// Начальная страница
            	TBL.iMsg:=0;				// Флаг ошибок загрузки
            ELSE
            	TBL.RowCount:=0;
            	TBL.RowSel:=-32768;			// Сброс выбора строки
            	TBL.PageNum:=0;				// Начальная страница
            	CASE iCount OF
            		0: TBL.iMsg:=0; 		// Список режимов пуст
            		-1: TBL.iMsg:=1; 		// Ошибка открытия файла
            		-2: TBL.iMsg:=2; 		// Носитель не смонтирован
            	END_CASE
            END_IF
        }
        OnMouseClick:  Dialog=DlgRegLoad, Parameters={pReg: ADR (REG_W), bExtEdit: FALSE}, OpenModal=True, OpenCentered=True
    RoundedRectangle (419,0 286x32), "%s", text variable: REG_W.Name
    Button (609,190 96x40), "Сохранить", text variable: REG_W.Name, input disabled if: NOT MMCMounted
        OnMouseClick: execute {
            IF RECORD_SAVE (ADR (REG_W)) THEN
            	iMsgShowDlg:=4;		// Запись успешно сохранена
            ELSE
            	iMsgShowDlg:=3;		// Ошибка сохранения
            END_IF
            CURRENT_PRG.bShowDialog:=TRUE;
        }
    Button (609,262 96x40), "Сохранить как", input disabled if: NOT MMCMounted
        OnMouseDown: execute { pTargetReg:=ADR (REG_W); }
        OnMouseClick:  Dialog=DlgKeyboard, Parameters={ilen: , sResult: REG_W.Name, bw: , bShift: , iStrLen: 63}, OpenModal=True, OpenCentered=True
    Button (609,46 96x40), "Редактор", text variable: REG_W.Name
        OnMouseClick: execute { SET_FRAME_INDEX (4); }
    Label (422,184 108x33), "Головка,Гц"
    RoundedRectangle (655,308 50x23), "%d", text variable: Asda.TorqueMin
    Label (602,312 55x21), "Tq min"
    Label (602,342 55x21), "Tq max"
    RoundedRectangle (655,338 50x23), "%d", text variable: Asda.TorqueMax
    Button (609,368 96x27), "Сбросить"
        OnMouseDown: execute { Asda.TorqueMin:=0; Asda.TorqueMax:=0; }
    RoundedRectangle (422,327 80x27), "ТЯУ, %", colour toggle: Dvp.Karet_si
END_VISUALIZATION

// Device/Application/Visu/DlgPids
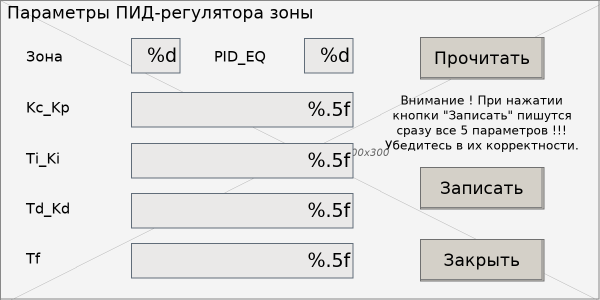
VISUALIZATION DlgPids  // 600x300
    Image (0,0 608x305), image: ImagePool.Dialog_win_7_600x300
    Button (420,37 124x42), "Прочитать"
        OnMouseClick: execute { Dvp.pid_read:=TRUE; }
    Button (420,239 124x42), "Закрыть"
        OnMouseClick:  Dialog=DlgPids, Result=OK, NumpadKeypadSet=True
    Label (4,3 373x19), "Параметры ПИД-регулятора зоны"
    Label (23,98 62x19), "Kc_Kp"
    RoundedRectangle (131,92 222x35), "%.5f", text variable: Dvp.Pids[Dvp.pid_index].Kc_Kp
        OnMouseClick: write the text variable via VisuDialogs.Numpad, min 0, max 1000, title "Пропорциональная часть"
    Label (23,149 62x19), "Ti_Ki"
    RoundedRectangle (131,143 222x35), "%.5f", text variable: Dvp.Pids[Dvp.pid_index].Ti_Ki
        OnMouseClick: write the text variable via VisuDialogs.Numpad, min 0, max 1000000, title "Интегральная часть"
    Label (23,199 62x19), "Td_Kd"
    RoundedRectangle (131,193 222x35), "%.5f", text variable: Dvp.Pids[Dvp.pid_index].Td_Kd
        OnMouseClick: write the text variable via VisuDialogs.Numpad, min 0, max 1000, title "Дифференциальная часть"
    RoundedRectangle (131,38 49x35), "%d", text variable: Dvp.zone_index
    Label (23,47 62x19), "Зона"
    Button (420,167 124x42), "Записать"
        OnMouseClick:  Dialog=DlgConfirm, Parameters={bDialogVar: Dvp.pid_write}, Selected={1: }, OpenModal=True, OpenCentered=True
    RoundedRectangle (304,38 49x35), "%d", text variable: Dvp.Pids[Dvp.pid_index].formula
        OnMouseClick: write the text variable via VisuDialogs.Numpad, min 0, max 1, format "Формула ПИД"
    Label (211,47 83x19), "PID_EQ"
    Label (23,249 62x19), "Tf"
    RoundedRectangle (131,243 222x35), "%.5f", text variable: Dvp.Pids[Dvp.pid_index].Tf
        OnMouseClick: write the text variable via VisuDialogs.Numpad, title "Пост.времени дифференцирования"
    Label (389,92 186x79), "Внимание ! При нажатии кнопки "Записать" пишутся сразу все 5 параметров !!! Убедитесь в их корректности."
END_VISUALIZATION

// Device/Application/Visu/VIS_SETTS_1
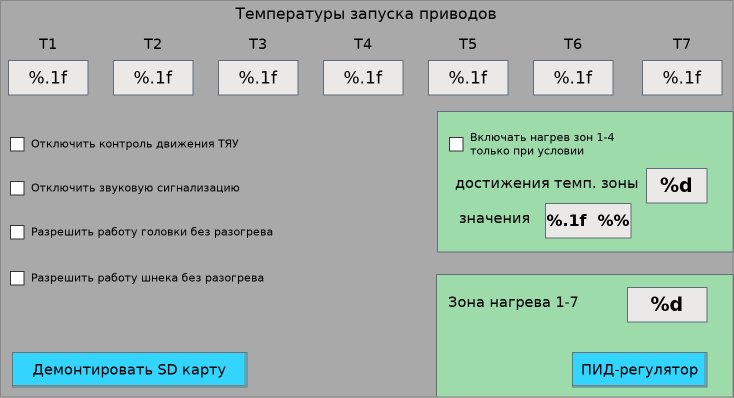
VISUALIZATION VIS_SETTS_1  // 734x398
    RoundedRectangle (436,274 298x123)
    RoundedRectangle (437,111 297x141)
    Label (219,3 294x28), "Температуры запуска приводов"
    RoundedRectangle (8,60 80x35), "%.1f", text variable: Setts.T_ZAP[0]
        OnMouseClick: write the text variable via VisuDialogs.Numpad, min T_ZAP_MIN, max T_ZAP_MAX, title "Температура зоны для запуска приводов"
    RoundedRectangle (323,60 80x35), "%.1f", text variable: Setts.T_ZAP[3]
        OnMouseClick: write the text variable via VisuDialogs.Numpad, min T_ZAP_MIN, max T_ZAP_MAX, title "Температура зоны для запуска приводов"
    RoundedRectangle (428,60 80x35), "%.1f", text variable: Setts.T_ZAP[4]
        OnMouseClick: write the text variable via VisuDialogs.Numpad, min T_ZAP_MIN, max T_ZAP_MAX, title "Температура зоны для запуска приводов"
    RoundedRectangle (533,60 80x35), "%.1f", text variable: Setts.T_ZAP[5]
        OnMouseClick: write the text variable via VisuDialogs.Numpad, min T_ZAP_MIN, max T_ZAP_MAX, title "Температура зоны для запуска приводов"
    RoundedRectangle (642,60 80x35), "%.1f", text variable: Setts.T_ZAP[6]
        OnMouseClick: write the text variable via VisuDialogs.Numpad, min T_ZAP_MIN, max T_ZAP_MAX, title "Температура зоны для запуска приводов"
    RoundedRectangle (218,60 80x35), "%.1f", text variable: Setts.T_ZAP[2]
        OnMouseClick: write the text variable via VisuDialogs.Numpad, min T_ZAP_MIN, max T_ZAP_MAX, title "Температура зоны для запуска приводов"
    RoundedRectangle (113,60 80x35), "%.1f", text variable: Setts.T_ZAP[1]
        OnMouseClick: write the text variable via VisuDialogs.Numpad, min T_ZAP_MIN, max T_ZAP_MAX, title "Температура зоны для запуска приводов"
    Label (8,34 80x25), "T1"
    Label (113,34 80x25), "T2"
    Label (218,34 80x25), "T3"
    Label (323,34 80x25), "T4"
    Label (428,34 80x25), "T5"
    Label (533,34 80x25), "T6"
    Label (642,34 80x25), "T7"
    Label (445,292 166x28), "Зона нагрева 1-7"
    Button (572,352 135x35), "ПИД-регулятор"
        OnMouseClick:  Dialog=DlgPids, Parameters={bDialogVar: b_dialog}, Selected={1: }, OpenModal=True, OpenCentered=True
    RoundedRectangle (627,287 80x35), "%d", text variable: Dvp.zone_index
        OnMouseClick: write the text variable via VisuDialogs.Numpad, min 1, max 7, title "Введите зону нагрева 1-7"
    Checkbox (8,169 412x38), "Отключить звуковую сигнализацию", variable: Setts.otkl_alarm_zvuk
    Checkbox (8,213 370x38), "Разрешить работу головки без разогрева", variable: Setts.use_servo_without_temp, input disabled if: TRUE
    Checkbox (8,259 412x38), "Разрешить работу шнека без разогрева", variable: Setts.use_shnek_without_temp, input disabled if: TRUE
    Checkbox (8,125 362x38), "Отключить контроль движения ТЯУ", variable: Setts.otkl_c_pulling
    Checkbox (447,123 243x42), "Включать нагрев зон 1-4 только при условии", variable: Setts.CondEnableZones1_4
    Label (452,173 201x28), "достижения темп. зоны"
    RoundedRectangle (646,168 61x35), "%d", text variable: Setts.CondIZone, input disabled if: NOT Setts.CondEnableZones1_4
        OnMouseClick: write the text variable via VisuDialogs.Numpad, min 5, max 7, title "Введите зону - образец 5-7"
    Label (456,208 78x29), "значения"
    RoundedRectangle (545,203 86x35), "%.1f %%", text variable: Setts.CondValue, input disabled if: NOT Setts.CondEnableZones1_4
        OnMouseClick: write the text variable via VisuDialogs.Numpad, min 0, max 100, title "Введите образцовое значение"
    Button (12,352 235x35), "Демонтировать SD карту"
        OnMouseClick: execute { bUnmount:=TRUE; }
END_VISUALIZATION

// Device/Application/Visu/VIS_SETTS_3
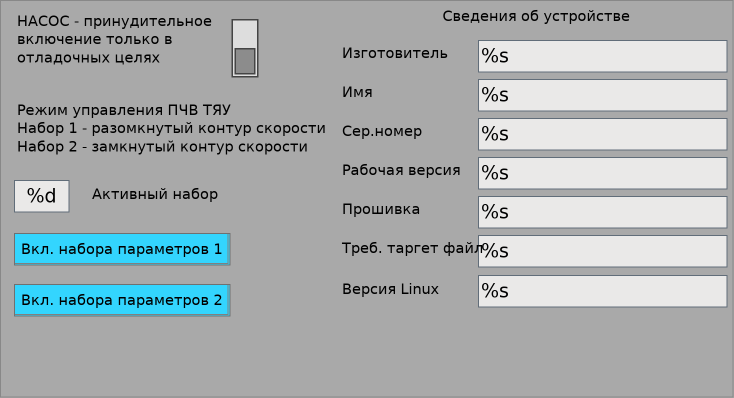
VISUALIZATION VIS_SETTS_3  // 734x398
    DipSwitch (216,19 58x58), variable: Dvp.Nasos_OTL, behaviour: TOGGLE, style: Switch-DipSwitch-Gray
    Label (14,11 194x77), "НАСОС - принудительное включение только в отладочных целях"
    Label (14,100 315x66), "Режим управления ПЧВ ТЯУ Набор 1 - разомкнутый контур скорости Набор 2 - замкнутый контур скорости"
    Button (14,233 216x32), "Вкл. набора параметров 1"
        OnMouseClick: execute {
            PARAM_SET:=1;
            // Запись режима управления тянущего устройства
            // Параметр 1 - Набор данных 1
            // 16#63 - адрес регистра активного набора параметров
            QueuePushReg (ADR (COM2_PRG.WR_REGS), ADR_PULLING, 16#63, ADR (PARAM_SET), 1);
        }
    Button (14,284 216x32), "Вкл. набора параметров 2"
        OnMouseClick: execute {
            PARAM_SET:=2;
            // Запись режима управления тянущего устройства
            // Параметр 1 - Набор данных 1
            // 16#63 - адрес регистра активного набора параметров
            QueuePushReg (ADR (COM2_PRG.WR_REGS), ADR_PULLING, 16#63, ADR (PARAM_SET), 1);
        }
    RoundedRectangle (14,180 55x32), "%d", text variable: Pulling.ActiveParamSet
    Label (89,184 134x27), "Активный набор"
    RoundedRectangle (478,196 249x32), "%s", text variable: Project.sFirmwareVersion
    Label (339,199 149x27), "Прошивка"
    RoundedRectangle (478,235 249x32), "%s", text variable: Project.sNeedTarget
    Label (339,238 150x27), "Треб. таргет файл"
    Label (339,279 150x27), "Версия Linux"
    RoundedRectangle (478,275 249x32), "%s", text variable: Project.sLinuxVersion
    Label (339,43 127x27), "Изготовитель"
    RoundedRectangle (478,40 249x32), "%s", text variable: Project.sVendor
    Label (346,6 381x27), "Сведения об устройстве"
    Label (339,82 114x27), "Имя"
    RoundedRectangle (478,79 249x32), "%s", text variable: Project.sName
    Label (339,121 114x27), "Сер.номер"
    RoundedRectangle (478,118 249x32), "%s", text variable: Project.sSerial
    Label (339,160 138x27), "Рабочая версия"
    RoundedRectangle (478,157 249x32), "%s", text variable: Project.sRuntime
END_VISUALIZATION

// Device/Application/Visu/DlgPulling
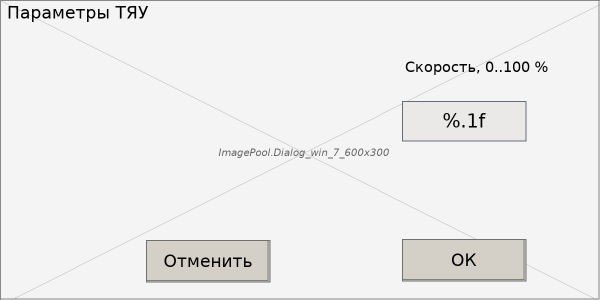
VISUALIZATION DlgPulling  // 600x300
VAR_IN_OUT
	fSpeed	: REAL;
END_VAR
    Image (0,0 608x305), image: ImagePool.Dialog_win_7_600x300
    Button (402,239 124x42), "ОК"
        OnMouseClick:  Dialog=DlgPulling, Result=OK, NumpadKeypadSet=True
    Label (4,3 186x19), "Параметры ТЯУ"
    Button (146,240 124x42), "Отменить"
        OnMouseClick:  Dialog=DlgPulling, Result=Cancel, NumpadKeypadSet=True
    RoundedRectangle (402,101 124x40), "%.1f", text variable: fSpeed
        OnMouseClick: write the text variable via VisuDialogs.Numpad, min SPEED_MIN, max SPEED_MAX, title "Скорость тянущего, %"
    Label (402,57 147x28), "Скорость, 0..100 %"
END_VISUALIZATION

// Device/Application/Visu/DlgTargetRegParams
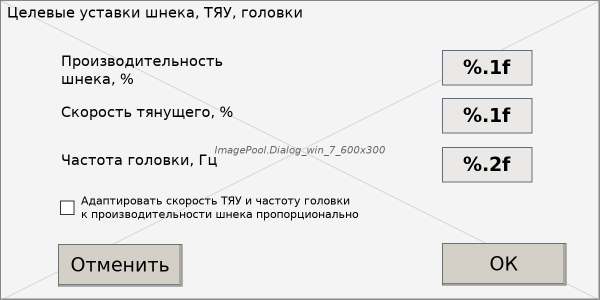
VISUALIZATION DlgTargetRegParams  // 600x300
VAR_INPUT
	fFreq	: REAL;
	fQm		: REAL;
	fSpeed	: REAL;
END_VAR

VAR
	fQm_old	: REAL;
	Adapted	: BOOL:=TRUE;
	bQm		: BOOL:=FALSE;
END_VAR
    Image (0,0 600x300), image: ImagePool.Dialog_win_7_600x300
    Button (442,243 124x42), "ОК"
        OnMouseClick:  Dialog=DlgTargetRegParams, Result=OK, NumpadKeypadSet=True
        OnMouseClick: execute {
            REG_W.Freq:=fFreq;
            REG_W.Qm:=fQm;
            REG_W.Speed:=fSpeed;
            AsdaSetParams ();
        }
    Label (4,3 341x19), "Целевые уставки шнека, ТЯУ, головки"
    Label (58,52 185x36), "Производительность шнека, %"
    Button (58,244 124x42), "Отменить"
        OnMouseClick:  Dialog=DlgTargetRegParams, Result=Cancel, NumpadKeypadSet=True
    RoundedRectangle (442,98 90x35), "%.1f", text variable: fSpeed
        OnMouseClick: write the text variable via VisuDialogs.Numpad, min SPEED_MIN, max SPEED_MAX, title "Скорость тянущего, %"
    Label (58,102 189x28), "Скорость тянущего, %"
    RoundedRectangle (442,50 90x35), "%.1f", text variable: fQm
        OnMouseClick: write the text variable via VisuDialogs.Numpad, min QM_MIN, max QM_MAX, title "Производительность шнека, %"
        OnMouseClick: execute {
            fQm_old:=fQm; // Производительность
            bQm:=TRUE;
        }
        OnDialogClosed: execute {
            IF bQm THEN
            	IF fQm <> fQm_old THEN
            		IF Adapted AND fQm_old <> 0 THEN
            			fSpeed:=MAX (SPEED_MIN, MIN (SPEED_MAX, fSpeed * fQm / fQm_old));
            			fFreq:=MAX (FREQ_MIN, MIN (FREQ_MAX, fFreq * fQm / fQm_old));
            		END_IF
            		fQm_old:=fQm;
            	END_IF
            	bQm:=FALSE;
            END_IF
        }
    Label (58,150 169x28), "Частота головки, Гц"
    RoundedRectangle (442,147 90x35), "%.2f", text variable: fFreq
        OnMouseClick: write the text variable via VisuDialogs.Numpad, min FREQ_MIN, max FREQ_MAX, title "Частота головки в Гц"
    Checkbox (58,189 461x37), "Адаптировать скорость ТЯУ и частоту головки к производительности шнека пропорционально", variable: Adapted
END_VISUALIZATION

// Device/Application/Visu/DlgConfirmAsdaCMD
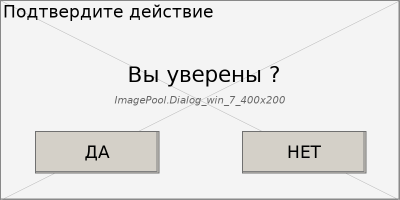
VISUALIZATION DlgConfirmAsdaCMD  // 400x200
VAR_INPUT
	fcmd: TWriteCmd;
END_VAR
    Image (0,0 400x200), image: ImagePool.Dialog_win_7_400x200
    Button (35,131 124x42), "ДА"
        OnMouseClick:  Dialog=DlgConfirmAsdaCMD, Result=OK, NumpadKeypadSet=True
        OnMouseClick: execute { AddWriteCmd (wcmd:=fcmd); }
    Button (242,131 124x42), "НЕТ"
        OnMouseClick:  Dialog=DlgConfirmAsdaCMD, Result=Cancel, NumpadKeypadSet=True
    Label (80,55 248x39), "Вы уверены ?"
    Label (0,0 248x23), "Подтвердите действие"
END_VISUALIZATION

// Device/Application/Visu/DlgRegLoad
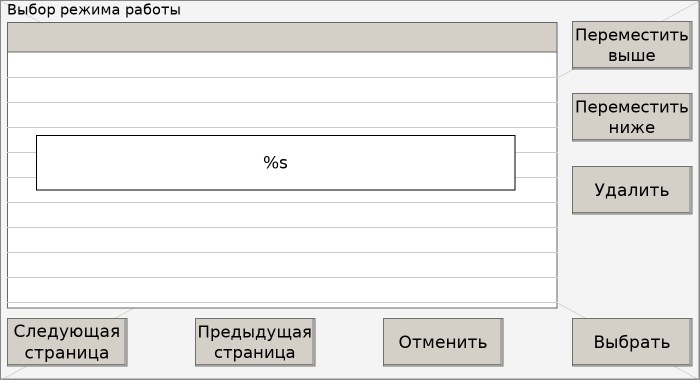
VISUALIZATION DlgRegLoad  // 700x380
VAR_INPUT
	pReg		: POINTER TO TReg;	// Указатель на режим, в который выбирается запись
	bExtEdit	: BOOL;				// Флаг расширенного редактирования
END_VAR

VAR
	
END_VAR
    Image (0,0 700x380), image: ImagePool.Dialog_win_7_700x380
    Button (572,318 120x48), "Выбрать", input disabled if: TBL.RowSel < 0
        OnMouseClick:  Dialog=DlgRegLoad, Result=OK, NumpadKeypadSet=True
        OnMouseClick: execute {
            pReg^:=TBL.Recs[TBL.RowSel]; // Записать выбранный режим редактирования
            // В случае если pReg является указателем на рабочий режим, то
            // запустим программу установки параметров сервопривода Asda
            IF (*IsRegValid (pReg) AND*) (pReg = ADR (REG_W)) THEN
            	AsdaSetParams ();
            END_IF
        }
    Label (4,0 341x19), "Выбор режима работы"
    Button (195,318 120x48), "Предыдущая страница", input disabled if: TBL.PageNum <= 0
        OnMouseClick: execute {
            TBL.PageNum:=TBL.PageNum-1;		// Уменьшим номер страницы
            TBL.RowCount:=RECS_SELECT (TBL.PageNum * TABLE_NUM_ROWS,
            	ADR (TBL.Recs), ADR (TBL.NumFileRecs));
            TBL.RowSel:=-32768;
        }
    Button (383,318 120x48), "Отменить"
        OnMouseClick:  Dialog=DlgRegLoad, Result=Cancel, NumpadKeypadSet=True
    Button (7,318 120x48), "Следующая страница", input disabled if: (TBL.PageNum*TABLE_NUM_ROWS+TBL.RowCount)>=TBL.NumFileRecs
        OnMouseClick: execute {
            TBL.PageNum:=TBL.PageNum + 1;		// Увеличим номер страницы
            TBL.RowCount:=RECS_SELECT (TBL.PageNum * TABLE_NUM_ROWS,
            	ADR (TBL.Recs), ADR (TBL.NumFileRecs));
            TBL.RowSel:=-32768;
        }
    Table (7,22 550x286), data array: TBL.Recs
        p1128707560: TBL.RowCount-1
        p1137915858: TBL.RowSel
        p3854506369: TBL.Recs[INDEX].Name
        p1892666644: TBL.Recs[INDEX].Desc
        p338671338: TBL.Recs[INDEX].TEMPS
        p2170511999: TBL.Recs[INDEX].T_MASS
        p3723444502: TBL.Recs[INDEX].T_CHIL
        p1218418051: TBL.Recs[INDEX].Period
        p2232123230: Имя
        p511219082: Т расп
        p1755163831: Т чил
        p4092479075: Qm,%
        p2237128397: ТЯУ,%
        p505689113: F, Гц
        p262371475: TBL.Recs[INDEX].Qm
        p4008173056: TBL.Recs[INDEX].Speed
        p2340480326: TBL.Recs[INDEX].Freq
    Rectangle (36,135 479x55), "%s", invisible if: TBL.RowCount>0, text list: 'FileTextList', text index: TBL.iMsg
    Button (572,166 120x48), "Удалить", input disabled if: NOT bExtEdit OR (TBL.RowSel < 0)
        OnMouseClick:  Dialog=DlgDeleteRec, Parameters={i_count: }, OpenModal=True, OpenCentered=True
    Button (572,21 120x48), "Переместить выше", input disabled if: NOT bExtEdit OR(TBL.RowSel<0)OR(TBL.NumFileRecs< 2)OR( (TBL.PageNum*TABLE_NUM_ROWS+TBL.RowSel)=0)
        OnMouseClick: execute {
            IF REC_EXCHANGE (TBL.PageNum * TABLE_NUM_ROWS + TBL.RowSel-1) THEN
            	TBL.RowSel:=TBL.RowSel-1;
            	IF TBL.RowSel < 0 THEN
            		TBL.RowSel:=TABLE_NUM_ROWS-1;
            		TBL.PageNum:=TBL.PageNum-1;
            	END_IF
            	TBL.RowCount:=RECS_SELECT (TBL.PageNum*TABLE_NUM_ROWS,
            		ADR (TBL.Recs), ADR (TBL.NumFileRecs));
            END_IF
        }
    Button (572,93 120x48), "Переместить ниже", input disabled if: NOT bExtEdit OR(TBL.RowSel<0)OR(TBL.NumFileRecs< 2)OR( (TBL.PageNum*TABLE_NUM_ROWS+TBL.RowSel)>=(TBL.NumFileRecs-1))
        OnMouseClick: execute {
            IF REC_EXCHANGE (TBL.PageNum * TABLE_NUM_ROWS + TBL.RowSel) THEN
            	TBL.RowSel:=TBL.RowSel + 1;
            	IF TBL.RowSel = TBL.RowCount THEN
            		TBL.RowSel:=0;
            		TBL.PageNum:=TBL.PageNum + 1;
            	END_IF
            	TBL.RowCount:=RECS_SELECT (TBL.PageNum * TABLE_NUM_ROWS,
            		ADR (TBL.Recs), ADR (TBL.NumFileRecs));
            END_IF
        }
END_VISUALIZATION

// Device/Application/Visu/DlgShow
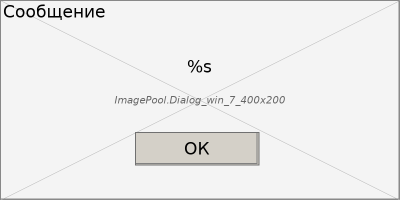
VISUALIZATION DlgShow  // 400x200
    Image (0,0 400x200), image: ImagePool.Dialog_win_7_400x200
    Button (135,132 124x33), "ОК"
        OnMouseClick:  Dialog=DlgShow, Result=OK, NumpadKeypadSet=True
    Label (0,0 248x22), "Сообщение"
    Textfield (9,28 381x77), "%s", text list: 'FileTextList', text index: iMsgShowDlg
END_VISUALIZATION

// Device/Application/Visu/DlgKeyboard
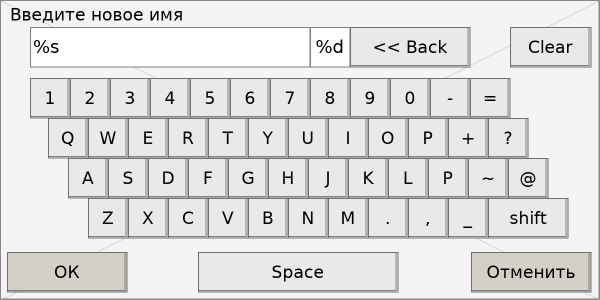
VISUALIZATION DlgKeyboard  // 600x300
VAR_INPUT
	sResult 	: STRING;				// Начальная и результирующая строка
	iStrLen		: INT;					// Максимальная длина строки
END_VAR
VAR
	bw			: BOOL:=FALSE;
	bShift		: BOOL:=FALSE;
	ilen		: INT;
END_VAR
    Image (0,0 600x300), image: ImagePool.Dialog_win_7_600x300
    Button (471,252 120x40), "Отменить"
        OnMouseClick:  Dialog=DlgKeyboard, Result=Cancel, NumpadKeypadSet=True
        OnMouseClick: execute { bw:=FALSE; bShift:=FALSE; }
    Label (7,4 354x21), "Введите новое имя"
    Button (7,252 120x40), "ОК", input disabled if: LEN ( OSCAT_BASIC.TRIM(sResult)) = 0
        OnMouseClick:  Dialog=DlgKeyboard, Result=OK, NumpadKeypadSet=True
        OnMouseClick: execute {
            bw:=FALSE;
            bShift:=FALSE;
            sResult:=OSCAT_BASIC.TRIM (sResult);	// Уберём ненужные пробелы
            REG_TEMP:=pTargetReg^;		// Записываем целевой режим во временный режим
            REG_TEMP.Name:=sResult;		// Записываем новое имя временного режима
            IF REC_NAME_EXISTS (sResult) THEN
            	// Запускаем диалог подтвержения перезаписи
            	CURRENT_PRG.bConfirmSaveAsDialog:=TRUE;
            ELSE
            	// Иначе записываем в файл
            	IF RECORD_SAVE (ADR (REG_TEMP)) THEN
            		iMsgShowDlg:=4;					// Запись успешно сохранена
            		pTargetReg^.Name:=sResult;		// Записывает новое имя в целевой режим
            	ELSE
            		iMsgShowDlg:=3;					// Ошибка сохранения
            		// В данном случае в целевом режиме останется старое имя
            	END_IF
            	// Запуск диалога сообщения
            	CURRENT_PRG.bShowDialog:=TRUE;
            END_IF
        }
    RoundedRectangle (30,27 280x40), "%s", text variable: sResult
    Button (30,78 40x40), "1"
        OnMouseDown: execute { KEYBOARD_STR ('1', ADR (sResult), ADR (bw), bShift, iStrLen); }
    Button (70,78 40x40), "2"
        OnMouseClick: execute { KEYBOARD_STR('2', ADR(sResult), ADR(bw), bShift, iStrLen); }
    Button (110,78 40x40), "3"
        OnMouseClick: execute { KEYBOARD_STR('3', ADR(sResult), ADR(bw), bShift, iStrLen); }
    Button (150,78 40x40), "4"
        OnMouseClick: execute { KEYBOARD_STR('4', ADR(sResult), ADR(bw), bShift, iStrLen); }
    Button (190,78 40x40), "5"
        OnMouseClick: execute { KEYBOARD_STR('5', ADR(sResult), ADR(bw), bShift, iStrLen); }
    Button (230,78 40x40), "6"
        OnMouseClick: execute { KEYBOARD_STR('6', ADR(sResult), ADR(bw), bShift, iStrLen); }
    Button (270,78 40x40), "7"
        OnMouseClick: execute { KEYBOARD_STR('7', ADR(sResult), ADR(bw), bShift, iStrLen); }
    Button (310,78 40x40), "8"
        OnMouseClick: execute { KEYBOARD_STR('8', ADR(sResult), ADR(bw), bShift, iStrLen); }
    Button (350,78 40x40), "9"
        OnMouseClick: execute { KEYBOARD_STR('9', ADR(sResult), ADR(bw), bShift, iStrLen); }
    Button (390,78 40x40), "0"
        OnMouseClick: execute { KEYBOARD_STR('0', ADR(sResult), ADR(bw), bShift, iStrLen); }
    Button (430,78 40x40), "-"
        OnMouseClick: execute { KEYBOARD_STR('-', ADR(sResult), ADR(bw), bShift, iStrLen); }
    Button (470,78 40x40), "="
        OnMouseClick: execute { KEYBOARD_STR('=', ADR(sResult), ADR(bw), bShift, iStrLen); }
    Button (48,118 40x40), "Q"
        OnMouseClick: execute { KEYBOARD_STR('Q', ADR(sResult), ADR(bw), bShift, iStrLen); }
    Button (88,118 40x40), "W"
        OnMouseClick: execute { KEYBOARD_STR('W', ADR(sResult), ADR(bw), bShift, iStrLen); }
    Button (128,118 40x40), "E"
        OnMouseClick: execute { KEYBOARD_STR('E', ADR(sResult), ADR(bw), bShift, iStrLen); }
    Button (168,118 40x40), "R"
        OnMouseClick: execute { KEYBOARD_STR('R', ADR(sResult), ADR(bw), bShift, iStrLen); }
    Button (208,118 40x40), "T"
        OnMouseClick: execute { KEYBOARD_STR('T', ADR(sResult), ADR(bw), bShift, iStrLen); }
    Button (248,118 40x40), "Y"
        OnMouseClick: execute { KEYBOARD_STR('Y', ADR(sResult), ADR(bw), bShift, iStrLen); }
    Button (288,118 40x40), "U"
        OnMouseClick: execute { KEYBOARD_STR('U', ADR(sResult), ADR(bw), bShift, iStrLen); }
    Button (328,118 40x40), "I"
        OnMouseClick: execute { KEYBOARD_STR('I', ADR(sResult), ADR(bw), bShift, iStrLen); }
    Button (368,118 40x40), "O"
        OnMouseClick: execute { KEYBOARD_STR('O', ADR(sResult), ADR(bw), bShift, iStrLen); }
    Button (408,118 40x40), "P"
        OnMouseClick: execute { KEYBOARD_STR('P', ADR(sResult), ADR(bw), bShift, iStrLen); }
    Button (448,118 40x40), "+"
        OnMouseClick: execute { KEYBOARD_STR('+', ADR(sResult), ADR(bw), bShift, iStrLen); }
    Button (488,118 40x40), "?"
        OnMouseClick: execute { KEYBOARD_STR('?', ADR(sResult), ADR(bw), bShift, iStrLen); }
    Button (68,158 40x40), "A"
        OnMouseClick: execute { KEYBOARD_STR ('A', ADR (sResult), ADR (bw), bShift, iStrLen); }
    Button (108,158 40x40), "S"
        OnMouseClick: execute { KEYBOARD_STR('S', ADR(sResult), ADR(bw), bShift, iStrLen); }
    Button (148,158 40x40), "D"
        OnMouseClick: execute { KEYBOARD_STR('D', ADR(sResult), ADR(bw), bShift, iStrLen); }
    Button (188,158 40x40), "F"
        OnMouseClick: execute { KEYBOARD_STR('F', ADR(sResult), ADR(bw), bShift, iStrLen); }
    Button (228,158 40x40), "G"
        OnMouseClick: execute { KEYBOARD_STR('G', ADR(sResult), ADR(bw), bShift, iStrLen); }
    Button (268,158 40x40), "H"
        OnMouseClick: execute { KEYBOARD_STR('H', ADR(sResult), ADR(bw), bShift, iStrLen); }
    Button (308,158 40x40), "J"
        OnMouseClick: execute { KEYBOARD_STR('J', ADR(sResult), ADR(bw), bShift, iStrLen); }
    Button (348,158 40x40), "K"
        OnMouseClick: execute { KEYBOARD_STR('K', ADR(sResult), ADR(bw), bShift, iStrLen); }
    Button (388,158 40x40), "L"
        OnMouseClick: execute { KEYBOARD_STR('L', ADR(sResult), ADR(bw), bShift, iStrLen); }
    Button (428,158 40x40), "P"
        OnMouseClick: execute { KEYBOARD_STR('P', ADR(sResult), ADR(bw), bShift, iStrLen); }
    Button (468,158 40x40), "~"
        OnMouseClick: execute { KEYBOARD_STR('~', ADR(sResult), ADR(bw), bShift, iStrLen); }
    Button (508,158 40x40), "@"
        OnMouseClick: execute { KEYBOARD_STR('@', ADR(sResult), ADR(bw), bShift, iStrLen); }
    Button (88,198 40x40), "Z"
        OnMouseClick: execute { KEYBOARD_STR('Z', ADR(sResult), ADR(bw), bShift, iStrLen); }
    Button (128,198 40x40), "X"
        OnMouseClick: execute { KEYBOARD_STR('X', ADR(sResult), ADR(bw), bShift, iStrLen); }
    Button (168,198 40x40), "C"
        OnMouseClick: execute { KEYBOARD_STR('C', ADR(sResult), ADR(bw), bShift, iStrLen); }
    Button (208,198 40x40), "V"
        OnMouseClick: execute { KEYBOARD_STR('V', ADR(sResult), ADR(bw), bShift, iStrLen); }
    Button (248,198 40x40), "B"
        OnMouseClick: execute { KEYBOARD_STR('B', ADR(sResult), ADR(bw), bShift, iStrLen); }
    Button (288,198 40x40), "N"
        OnMouseClick: execute { KEYBOARD_STR('N', ADR(sResult), ADR(bw), bShift, iStrLen); }
    Button (328,198 40x40), "M"
        OnMouseClick: execute { KEYBOARD_STR('M', ADR(sResult), ADR(bw), bShift, iStrLen); }
    Button (368,198 40x40), "."
        OnMouseClick: execute { KEYBOARD_STR('.', ADR(sResult), ADR(bw), bShift, iStrLen); }
    Button (408,198 40x40), ","
        OnMouseClick: execute { KEYBOARD_STR(',', ADR(sResult), ADR(bw), bShift, iStrLen); }
    Button (448,198 40x40), "_"
        OnMouseClick: execute { KEYBOARD_STR('_', ADR(sResult), ADR(bw), bShift, iStrLen); }
    Button (488,198 80x40), "shift", colour toggle: bShift
        OnMouseClick: execute { bShift:=NOT bShift; }
    RoundedRectangle (310,27 40x40), "%d", text variable: LEN (sResult)
    Button (198,252 200x40), "Space"
        OnMouseClick: execute { KEYBOARD_STR (' ', ADR (sResult), ADR (bw), bShift, iStrLen); }
    Button (510,27 81x40), "Clear"
        OnMouseClick: execute { bw:=TRUE; sResult:=''; }
    Button (350,27 120x40), "<< Back"
        OnMouseClick: execute {
            IF LEN (sResult) > 0 THEN
            	sResult:=DELETE (sResult, 1, LEN (sResult));
            END_IF
            bw:=TRUE;
        }
END_VISUALIZATION

// Device/Application/Visu/DlgConfirmSaveAS
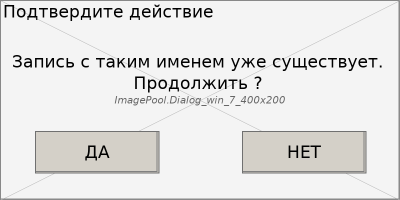
VISUALIZATION DlgConfirmSaveAS  // 400x200
VAR_IN_OUT
	bDialogVar	: BOOL;
END_VAR
    Image (0,0 400x200), image: ImagePool.Dialog_win_7_400x200
    Button (35,131 124x42), "ДА"
        OnMouseClick:  Dialog=DlgConfirmSaveAS, Result=OK, NumpadKeypadSet=True
        OnMouseClick: execute {
            IF RECORD_SAVE (ADR (REG_TEMP)) THEN // REG_TEMP сформирована ранее
            	pTargetReg^.Name:=REG_TEMP.Name;
            	iMsgShowDlg:=4;		// Успешно
            ELSE
            	iMsgShowDlg:=3;		// Ошибка сохранения
            END_IF
            // Запуск диалга сообщения
            CURRENT_PRG.bShowDialog:=TRUE;
        }
    Button (242,131 124x42), "НЕТ"
        OnMouseClick:  Dialog=DlgConfirmSaveAS, Result=Cancel, NumpadKeypadSet=True
    Label (7,41 382x63), "Запись с таким именем уже существует. Продолжить ?"
    Label (0,0 248x27), "Подтвердите действие"
END_VISUALIZATION

// Device/Application/Visu/VIS_EDITOR
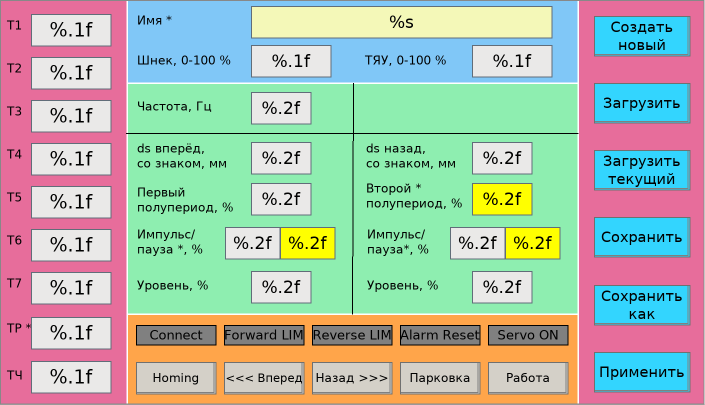
VISUALIZATION VIS_EDITOR  // 705x405
VAR_IN_OUT

END_VAR

